RoboDK station: Config_2.rdk

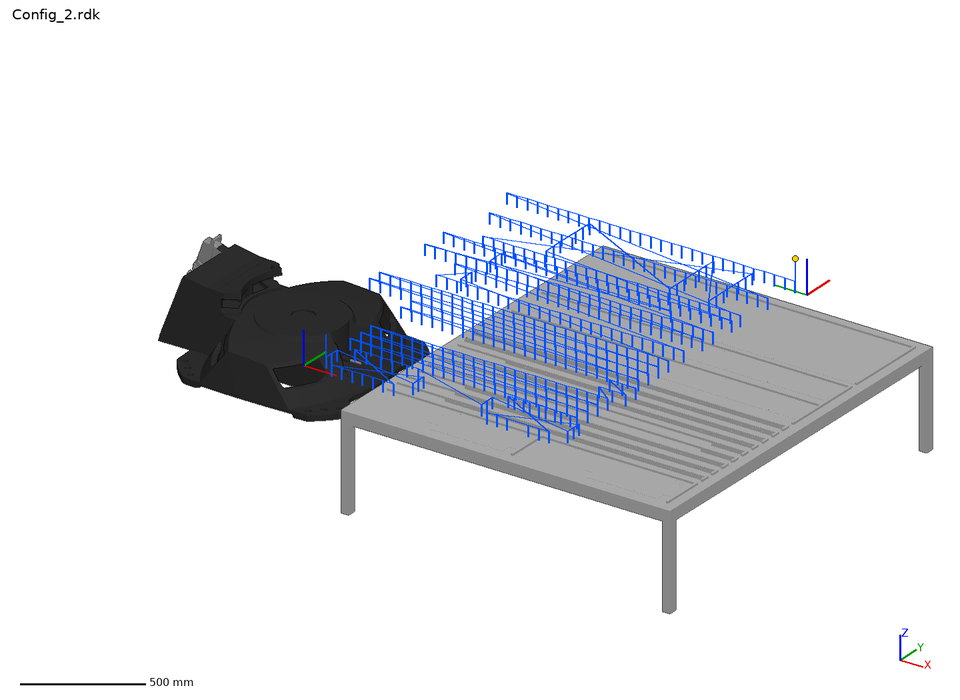
[picture v0: the station drawn from its stored meshes, robots at their saved joint values, targets as dots, program paths as lines]
Station Config_2 (saved by RoboDK 5.2.3). Poses are relative to the parent item; angles as X-Y-Z fixed-axis rotations.
  - frame KUKA KR 210 R2700 extra Base at (0, 0, 0) mm
    - robot KUKA KR 210 R2700 extra: 6 axes, payload 210 kg, reach 2696 mm, repeatability 0.06 mm, weight 1068 kg
        joint limits [-185, -140, -120, -350, -125, -350] to [185, -5, 155, 350, 125, 350]; home [0, -90, 90, 0, 0, 0]; saved at [44.26, -78.74, 122.767, 234.505, 59.006, -215.831]
      - tool Spindle, TCP at (278.6, 0, 88) mm, rotated rx 0 ry 90 rz 0 deg, size 85 x 346.5 x 128 mm
  - frame Corner First Plate at (1872.67, 817.07, 510.8) mm, rotated rx 0 ry 0 rz 90 deg
  - object Table 2 at (1700, -800, 455) mm, rotated rx 0 ry 0 rz 90 deg, size 1820 x 1600 x 475 mm, geometry from Table 2.stl
  - object Config_2 at (2495, 660, 510.8) mm, rotated rx 0 ry 0 rz 90 deg
  - machining project Path1 settings: rotZ(0) | rotX(0)*rotY(0) | rotz(0) | onStart | onPathStart | onApproach | onPoint | onRetract | onFinish | SetRPM(%1) | SetTool(%1) | Extruder(%1) | default | default | OutOnMov(%1) | OutOffMov(%1) | onPathFinish | M_RunCode(%1)
  - program Path1 (1338 instructions, listed below)
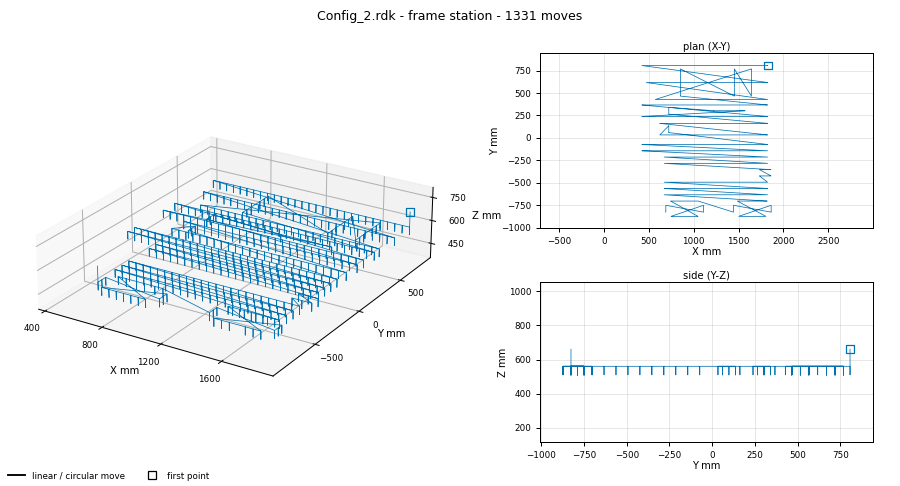
[picture p0: tool path of Config_2.rdk in frame station, 1331 of 1331 moves have a stored position in this frame; points joined in program order, loops and branches not executed]

--- program Path1 (robot KUKA KR 210 R2700 extra) ---
  Smooth(1)
  Set speed (1000.0 mm/s)
  Set Ref.: Corner First Plate
  Set Tool: Spindle
  Show Spindle
  MoveJ 1 to (-10.8, 50, 150) mm, rotated rx 180 ry 0 rz 90 deg; joints [-16.861, -44.669, 69.656, 144.341, 29.838, -148.103]
  MoveL 2 to (-10.8, 50, 150) mm, rotated rx 180 ry 0 rz 90 deg; joints [-16.861, -44.669, 69.656, 144.341, 29.838, -148.103]
  MoveL 3 to (-10.8, 50, 50) mm, rotated rx 180 ry 0 rz 90 deg; joints [-16.861, -42.157, 70.591, 147.522, 32.695, -151.823]
  MoveL 4 to (-10.8, 50, 50) mm, rotated rx 180 ry 0 rz 90 deg; joints [-16.861, -42.157, 70.591, 147.522, 32.695, -151.823]
  Set speed (150.0 mm/s)
  MoveL 5 to (-10.8, 50, -0.5) mm, rotated rx -180 ry 0 rz 90 deg; joints [-16.861, -40.791, 70.897, 148.859, 34.116, -153.424]
  MoveL 6 to (-10.8, 50, 50) mm, rotated rx 180 ry 0 rz 90 deg; joints [-16.861, -42.157, 70.591, 147.522, 32.695, -151.823]
  MoveL 7 to (-10.8, 100, 50) mm, rotated rx -180 ry 0 rz 90 deg; joints [-17.24, -44.27, 74.43, 148.298, 34.333, -152.976]
  MoveL 8 to (-10.8, 100, -0.5) mm, rotated rx -180 ry 0 rz 90 deg; joints [-17.24, -42.862, 74.73, 149.554, 35.795, -154.51]
  MoveL 9 to (-10.8, 100, 50) mm, rotated rx -180 ry 0 rz 90 deg; joints [-17.24, -44.27, 74.43, 148.298, 34.333, -152.976]
  MoveL 10 to (-10.8, 150, 50) mm, rotated rx -180 ry 0 rz 90 deg; joints [-17.637, -46.308, 78.104, 148.894, 35.906, -153.954]
  MoveL 11 to (-10.8, 150, -0.5) mm, rotated rx 180 ry 0 rz 90 deg; joints [-17.637, -44.857, 78.4, 150.085, 37.411, -155.439]
  MoveL 12 to (-10.8, 150, 50) mm, rotated rx -180 ry 0 rz 90 deg; joints [-17.637, -46.308, 78.104, 148.894, 35.906, -153.954]
  MoveL 13 to (-10.8, 200, 50) mm, rotated rx 180 ry 0 rz 90 deg; joints [-18.051, -48.282, 81.634, 149.341, 37.421, -154.79]
  MoveL 14 to (-10.8, 200, -0.5) mm, rotated rx -180 ry 0 rz 90 deg; joints [-18.051, -46.786, 81.927, 150.481, 38.968, -156.24]
  MoveL 15 to (-10.8, 200, 50) mm, rotated rx 180 ry 0 rz 90 deg; joints [-18.051, -48.282, 81.634, 149.341, 37.421, -154.79]
  MoveL 16 to (-10.8, 250, 50) mm, rotated rx 180 ry 0 rz 90 deg; joints [-18.485, -50.201, 85.037, 149.663, 38.882, -155.508]
  MoveL 17 to (-10.8, 250, -0.5) mm, rotated rx -180 ry 0 rz 90 deg; joints [-18.485, -48.66, 85.329, 150.761, 40.473, -156.934]
  MoveL 18 to (-10.8, 250, 50) mm, rotated rx 180 ry 0 rz 90 deg; joints [-18.485, -50.201, 85.037, 149.663, 38.882, -155.508]
  MoveL 19 to (-10.8, 300, 50) mm, rotated rx -180 ry 0 rz 90 deg; joints [-18.939, -52.073, 88.328, 149.877, 40.293, -156.128]
  MoveL 20 to (-10.8, 300, -0.5) mm, rotated rx 180 ry 0 rz 90 deg; joints [-18.939, -50.484, 88.62, 150.941, 41.929, -157.54]
  MoveL 21 to (-10.8, 300, 50) mm, rotated rx -180 ry 0 rz 90 deg; joints [-18.939, -52.073, 88.328, 149.877, 40.293, -156.128]
  MoveL 22 to (-10.8, 350, 50) mm, rotated rx 180 ry 0 rz 90 deg; joints [-19.415, -53.906, 91.518, 149.994, 41.659, -156.663]
  MoveL 23 to (-10.8, 350, -0.5) mm, rotated rx 180 ry 0 rz 90 deg; joints [-19.415, -52.267, 91.81, 151.032, 43.339, -158.069]
  MoveL 24 to (-10.8, 350, 50) mm, rotated rx 180 ry 0 rz 90 deg; joints [-19.415, -53.906, 91.518, 149.994, 41.659, -156.663]
  MoveL 25 to (-10.8, 400, 50) mm, rotated rx 180 ry 0 rz 90 deg; joints [-19.914, -55.704, 94.616, 150.026, 42.981, -157.123]
  MoveL 26 to (-10.8, 400, -0.5) mm, rotated rx -180 ry 0 rz 90 deg; joints [-19.914, -54.013, 94.91, 151.042, 44.709, -158.532]
  MoveL 27 to (-10.8, 400, 50) mm, rotated rx 180 ry 0 rz 90 deg; joints [-19.914, -55.704, 94.616, 150.026, 42.981, -157.123]
  MoveL 28 to (-10.8, 450, 50) mm, rotated rx 180 ry 0 rz 90 deg; joints [-20.439, -57.473, 97.631, 149.977, 44.262, -157.517]
  MoveL 29 to (-10.8, 450, -0.5) mm, rotated rx 180 ry 0 rz 90 deg; joints [-20.439, -55.727, 97.926, 150.978, 46.038, -158.936]
  MoveL 30 to (-10.8, 450, 50) mm, rotated rx 180 ry 0 rz 90 deg; joints [-20.439, -57.473, 97.631, 149.977, 44.262, -157.517]
  MoveL 31 to (-10.8, 500, 50) mm, rotated rx -180 ry 0 rz 90 deg; joints [-20.991, -59.217, 100.569, 149.854, 45.504, -157.852]
  MoveL 32 to (-10.8, 500, -0.5) mm, rotated rx 180 ry 0 rz 90 deg; joints [-20.991, -57.414, 100.867, 150.844, 47.331, -159.288]
  MoveL 33 to (-10.8, 500, 50) mm, rotated rx -180 ry 0 rz 90 deg; joints [-20.991, -59.217, 100.569, 149.854, 45.504, -157.852]
  MoveL 34 to (-10.8, 550, 50) mm, rotated rx 180 ry 0 rz 90 deg; joints [-21.572, -60.942, 103.435, 149.66, 46.709, -158.133]
  MoveL 35 to (-10.8, 550, -0.5) mm, rotated rx 180 ry 0 rz 90 deg; joints [-21.572, -59.078, 103.738, 150.643, 48.588, -159.592]
  MoveL 36 to (-10.8, 550, 50) mm, rotated rx 180 ry 0 rz 90 deg; joints [-21.572, -60.942, 103.435, 149.66, 46.709, -158.133]
  MoveL 37 to (-10.8, 600, 50) mm, rotated rx 180 ry 0 rz 90 deg; joints [-22.185, -62.649, 106.236, 149.397, 47.878, -158.362]
  MoveL 38 to (-10.8, 600, -0.5) mm, rotated rx 180 ry 0 rz 90 deg; joints [-22.185, -60.721, 106.543, 150.377, 49.812, -159.851]
  MoveL 39 to (-10.8, 600, 50) mm, rotated rx 180 ry 0 rz 90 deg; joints [-22.185, -62.649, 106.236, 149.397, 47.878, -158.362]
  MoveL 40 to (-10.8, 650, 50) mm, rotated rx 180 ry 0 rz 90 deg; joints [-22.832, -64.344, 108.975, 149.067, 49.013, -158.542]
  MoveL 41 to (-10.8, 650, -0.5) mm, rotated rx 180 ry 0 rz 90 deg; joints [-22.832, -62.348, 109.287, 150.048, 51.003, -160.069]
  MoveL 42 to (-10.8, 650, 50) mm, rotated rx 180 ry 0 rz 90 deg; joints [-22.832, -64.344, 108.975, 149.067, 49.013, -158.542]
  MoveL 43 to (-10.8, 700, 50) mm, rotated rx -180 ry 0 rz 90 deg; joints [-23.515, -66.029, 111.655, 148.669, 50.113, -158.676]
  MoveL 44 to (-10.8, 700, -0.5) mm, rotated rx 180 ry 0 rz 90 deg; joints [-23.515, -63.961, 111.973, 149.655, 52.163, -160.247]
  MoveL 45 to (-10.8, 700, 50) mm, rotated rx -180 ry 0 rz 90 deg; joints [-23.515, -66.029, 111.655, 148.669, 50.113, -158.676]
  MoveL 46 to (-10.8, 750, 50) mm, rotated rx 180 ry 0 rz 90 deg; joints [-24.238, -67.708, 114.279, 148.204, 51.181, -158.763]
  MoveL 47 to (-10.8, 750, -0.5) mm, rotated rx 180 ry 0 rz 90 deg; joints [-24.238, -65.564, 114.604, 149.198, 53.292, -160.386]
  MoveL 48 to (-10.8, 750, 50) mm, rotated rx 180 ry 0 rz 90 deg; joints [-24.238, -67.708, 114.279, 148.204, 51.181, -158.763]
  MoveL 49 to (-10.8, 800, 50) mm, rotated rx -180 ry 0 rz 90 deg; joints [-25.003, -69.384, 116.85, 147.669, 52.216, -158.805]
  MoveL 50 to (-10.8, 800, -0.5) mm, rotated rx 180 ry 0 rz 90 deg; joints [-25.003, -67.159, 117.183, 148.675, 54.391, -160.488]
  MoveL 51 to (-10.8, 800, 50) mm, rotated rx -180 ry 0 rz 90 deg; joints [-25.003, -69.384, 116.85, 147.669, 52.216, -158.805]
  MoveL 52 to (-10.8, 850, 50) mm, rotated rx -180 ry 0 rz 90 deg; joints [-25.816, -71.061, 119.369, 147.064, 53.22, -158.799]
  MoveL 53 to (-10.8, 850, -0.5) mm, rotated rx 180 ry 0 rz 90 deg; joints [-25.816, -68.749, 119.711, 148.085, 55.46, -160.551]
  MoveL 54 to (-10.8, 850, 50) mm, rotated rx -180 ry 0 rz 90 deg; joints [-25.816, -71.061, 119.369, 147.064, 53.22, -158.799]
  MoveL 55 to (-10.8, 900, 50) mm, rotated rx 180 ry 0 rz 90 deg; joints [-26.678, -72.742, 121.838, 146.383, 54.192, -158.746]
  MoveL 56 to (-10.8, 900, -0.5) mm, rotated rx -180 ry 0 rz 90 deg; joints [-26.678, -70.337, 122.19, 147.424, 56.501, -160.575]
  MoveL 57 to (-10.8, 900, 50) mm, rotated rx 180 ry 0 rz 90 deg; joints [-26.678, -72.742, 121.838, 146.383, 54.192, -158.746]
  MoveL 58 to (-10.8, 950, 50) mm, rotated rx -180 ry 0 rz 90 deg; joints [-27.596, -74.43, 124.259, 145.626, 55.132, -158.641]
  MoveL 59 to (-10.8, 950, -0.5) mm, rotated rx -180 ry 0 rz 90 deg; joints [-27.596, -71.926, 124.621, 146.689, 57.513, -160.559]
  MoveL 60 to (-10.8, 950, 50) mm, rotated rx -180 ry 0 rz 90 deg; joints [-27.596, -74.43, 124.259, 145.626, 55.132, -158.641]
  MoveL 61 to (-10.8, 1000, 50) mm, rotated rx 180 ry 0 rz 90 deg; joints [-28.574, -76.128, 126.631, 144.786, 56.043, -158.484]
  MoveL 62 to (-10.8, 1000, -0.5) mm, rotated rx 180 ry 0 rz 90 deg; joints [-28.574, -73.519, 127.005, 145.877, 58.497, -160.501]
  MoveL 63 to (-10.8, 1000, 50) mm, rotated rx 180 ry 0 rz 90 deg; joints [-28.574, -76.128, 126.631, 144.786, 56.043, -158.484]
  MoveL 64 to (-10.8, 1050, 50) mm, rotated rx -180 ry 0 rz 90 deg; joints [-29.617, -77.842, 128.955, 143.858, 56.923, -158.269]
  MoveL 65 to (-10.8, 1050, -0.5) mm, rotated rx 180 ry 0 rz 90 deg; joints [-29.617, -75.119, 129.342, 144.981, 59.453, -160.398]
  MoveL 66 to (-10.8, 1050, 50) mm, rotated rx -180 ry 0 rz 90 deg; joints [-29.617, -77.842, 128.955, 143.858, 56.923, -158.269]
  MoveL 67 to (-10.8, 1100, 50) mm, rotated rx 180 ry 0 rz 90 deg; joints [-30.732, -79.573, 131.231, 142.838, 57.775, -157.992]
  MoveL 68 to (-10.8, 1100, -0.5) mm, rotated rx -180 ry 0 rz 90 deg; joints [-30.732, -76.729, 131.632, 143.997, 60.382, -160.246]
  MoveL 69 to (-10.8, 1100, 50) mm, rotated rx 180 ry 0 rz 90 deg; joints [-30.732, -79.573, 131.231, 142.838, 57.775, -157.992]
  MoveL 70 to (-10.8, 1150, 50) mm, rotated rx 180 ry 0 rz 90 deg; joints [-31.924, -81.327, 133.457, 141.718, 58.599, -157.647]
  MoveL 71 to (-10.8, 1150, -0.5) mm, rotated rx 180 ry 0 rz 90 deg; joints [-31.924, -78.352, 133.874, 142.918, 61.284, -160.042]
  MoveL 72 to (-10.8, 1150, 50) mm, rotated rx 180 ry 0 rz 90 deg; joints [-31.924, -81.327, 133.457, 141.718, 58.599, -157.647]
  MoveL 73 to (-10.8, 1200, 50) mm, rotated rx 180 ry 0 rz 90 deg; joints [-33.202, -83.108, 135.634, 140.49, 59.397, -157.227]
  MoveL 74 to (-10.8, 1200, -0.5) mm, rotated rx 180 ry 0 rz 90 deg; joints [-33.202, -79.993, 136.068, 141.737, 62.161, -159.78]
  MoveL 75 to (-10.8, 1200, 50) mm, rotated rx 180 ry 0 rz 90 deg; joints [-33.202, -83.108, 135.634, 140.49, 59.397, -157.227]
  MoveL 76 to (-10.8, 1250, 50) mm, rotated rx -180 ry 0 rz 90 deg; joints [-34.574, -84.92, 137.758, 139.147, 60.172, -156.726]
  MoveL 77 to (-10.8, 1250, -0.5) mm, rotated rx -180 ry 0 rz 90 deg; joints [-34.574, -81.654, 138.211, 140.446, 63.014, -159.455]
  MoveL 78 to (-10.8, 1250, 50) mm, rotated rx -180 ry 0 rz 90 deg; joints [-34.574, -84.92, 137.758, 139.147, 60.172, -156.726]
  MoveL 79 to (-10.8, 1300, 50) mm, rotated rx 180 ry 0 rz 90 deg; joints [-36.047, -86.767, 139.828, 137.68, 60.929, -156.133]
  MoveL 80 to (-10.8, 1300, -0.5) mm, rotated rx 180 ry 0 rz 90 deg; joints [-36.047, -83.339, 140.302, 139.037, 63.846, -159.059]
  MoveL 81 to (-10.8, 1300, 50) mm, rotated rx 180 ry 0 rz 90 deg; joints [-36.047, -86.767, 139.828, 137.68, 60.929, -156.133]
  MoveL 82 to (-10.8, 1350, 50) mm, rotated rx 180 ry 0 rz 90 deg; joints [-37.633, -88.655, 141.842, 136.078, 61.671, -155.439]
  MoveL 83 to (-10.8, 1350, -0.5) mm, rotated rx 180 ry 0 rz 90 deg; joints [-37.633, -85.052, 142.339, 137.499, 64.659, -158.585]
  MoveL 84 to (-10.8, 1350, 50) mm, rotated rx 180 ry 0 rz 90 deg; joints [-37.633, -88.655, 141.842, 136.078, 61.671, -155.439]
  MoveL 85 to (-10.8, 1400, 50) mm, rotated rx -180 ry 0 rz 90 deg; joints [-39.341, -90.587, 143.795, 134.333, 62.407, -154.634]
  MoveL 86 to (-10.8, 1400, -0.5) mm, rotated rx 180 ry 0 rz 90 deg; joints [-39.341, -86.798, 144.317, 135.822, 65.461, -158.023]
  MoveL 87 to (-10.8, 1400, 50) mm, rotated rx -180 ry 0 rz 90 deg; joints [-39.341, -90.587, 143.795, 134.333, 62.407, -154.634]
  MoveL 88 to (-10.8, 1450, 50) mm, rotated rx 180 ry 0 rz 90 deg; joints [-41.184, -92.567, 145.684, 132.434, 63.147, -153.707]
  MoveL 89 to (-10.8, 1450, -0.5) mm, rotated rx -180 ry 0 rz 90 deg; joints [-41.184, -88.578, 146.233, 133.998, 66.256, -157.364]
  MoveL 90 to (-10.8, 1450, 50) mm, rotated rx 180 ry 0 rz 90 deg; joints [-41.184, -92.567, 145.684, 132.434, 63.147, -153.707]
  MoveL 91 to (-200, 50, 50) mm, rotated rx -180 ry 0 rz 90 deg; joints [-12.12, -44.252, 74.397, 156.847, 32.277, -160.122]
  MoveL 92 to (-200, 50, -0.5) mm, rotated rx -180 ry 0 rz 90 deg; joints [-12.12, -42.844, 74.697, 157.857, 33.853, -161.328]
  MoveL 93 to (-200, 50, 50) mm, rotated rx -180 ry 0 rz 90 deg; joints [-12.12, -44.252, 74.397, 156.847, 32.277, -160.122]
  MoveL 94 to (-200, 100, 50) mm, rotated rx 180 ry 0 rz 90 deg; joints [-12.401, -46.339, 78.159, 157.362, 33.914, -160.91]
  MoveL 95 to (-200, 100, -0.5) mm, rotated rx 180 ry 0 rz 90 deg; joints [-12.401, -44.887, 78.455, 158.313, 35.532, -162.067]
  MoveL 96 to (-200, 100, 50) mm, rotated rx 180 ry 0 rz 90 deg; joints [-12.401, -46.339, 78.159, 157.362, 33.914, -160.91]
  MoveL 97 to (-200, 150, 50) mm, rotated rx 180 ry 0 rz 90 deg; joints [-12.695, -48.361, 81.776, 157.752, 35.481, -161.577]
  MoveL 98 to (-200, 150, -0.5) mm, rotated rx -180 ry 0 rz 90 deg; joints [-12.695, -46.864, 82.069, 158.657, 37.144, -162.699]
  MoveL 99 to (-200, 150, 50) mm, rotated rx 180 ry 0 rz 90 deg; joints [-12.695, -48.361, 81.776, 157.752, 35.481, -161.577]
  MoveL 100 to (-200, 200, 50) mm, rotated rx -180 ry 0 rz 90 deg; joints [-13.003, -50.329, 85.264, 158.038, 36.986, -162.145]
  MoveL 101 to (-200, 200, -0.5) mm, rotated rx -180 ry 0 rz 90 deg; joints [-13.003, -48.785, 85.556, 158.905, 38.694, -163.244]
  MoveL 102 to (-200, 200, 50) mm, rotated rx -180 ry 0 rz 90 deg; joints [-13.003, -50.329, 85.264, 158.038, 36.986, -162.145]
  MoveL 103 to (-200, 250, 50) mm, rotated rx -180 ry 0 rz 90 deg; joints [-13.326, -52.251, 88.639, 158.234, 38.432, -162.632]
  MoveL 104 to (-200, 250, -0.5) mm, rotated rx 180 ry 0 rz 90 deg; joints [-13.326, -50.658, 88.93, 159.072, 40.188, -163.715]
  MoveL 105 to (-200, 250, 50) mm, rotated rx -180 ry 0 rz 90 deg; joints [-13.326, -52.251, 88.639, 158.234, 38.432, -162.632]
  MoveL 106 to (-200, 300, 50) mm, rotated rx 180 ry 0 rz 90 deg; joints [-13.665, -54.134, 91.913, 158.353, 39.825, -163.049]
  MoveL 107 to (-200, 300, -0.5) mm, rotated rx 180 ry 0 rz 90 deg; joints [-13.665, -52.489, 92.205, 159.169, 41.63, -164.124]
  MoveL 108 to (-200, 300, 50) mm, rotated rx 180 ry 0 rz 90 deg; joints [-13.665, -54.134, 91.913, 158.353, 39.825, -163.049]
  MoveL 109 to (-200, 350, 50) mm, rotated rx 180 ry 0 rz 90 deg; joints [-14.022, -55.984, 95.096, 158.403, 41.167, -163.405]
  MoveL 110 to (-200, 350, -0.5) mm, rotated rx -180 ry 0 rz 90 deg; joints [-14.022, -54.285, 95.39, 159.201, 43.025, -164.48]
  MoveL 111 to (-200, 350, 50) mm, rotated rx 180 ry 0 rz 90 deg; joints [-14.022, -55.984, 95.096, 158.403, 41.167, -163.405]
  MoveL 112 to (-200, 400, 50) mm, rotated rx -180 ry 0 rz 90 deg; joints [-14.397, -57.808, 98.197, 158.389, 42.461, -163.709]
  MoveL 113 to (-200, 400, -0.5) mm, rotated rx 180 ry 0 rz 90 deg; joints [-14.397, -56.051, 98.494, 159.174, 44.374, -164.79]
  MoveL 114 to (-200, 400, 50) mm, rotated rx -180 ry 0 rz 90 deg; joints [-14.397, -57.808, 98.197, 158.389, 42.461, -163.709]
  MoveL 115 to (-200, 450, 50) mm, rotated rx 180 ry 0 rz 90 deg; joints [-14.792, -59.609, 101.223, 158.316, 43.709, -163.964]
  MoveL 116 to (-200, 450, -0.5) mm, rotated rx 180 ry 0 rz 90 deg; joints [-14.792, -57.793, 101.523, 159.093, 45.681, -165.057]
  MoveL 117 to (-200, 450, 50) mm, rotated rx 180 ry 0 rz 90 deg; joints [-14.792, -59.609, 101.223, 158.316, 43.709, -163.964]
  MoveL 118 to (-200, 500, 50) mm, rotated rx 180 ry 0 rz 90 deg; joints [-15.209, -61.394, 104.181, 158.187, 44.913, -164.175]
  MoveL 119 to (-200, 500, -0.5) mm, rotated rx 180 ry 0 rz 90 deg; joints [-15.209, -59.513, 104.485, 158.96, 46.946, -165.286]
  MoveL 120 to (-200, 500, 50) mm, rotated rx 180 ry 0 rz 90 deg; joints [-15.209, -61.394, 104.181, 158.187, 44.913, -164.175]
  MoveL 121 to (-200, 550, 50) mm, rotated rx 180 ry 0 rz 90 deg; joints [-15.65, -63.166, 107.075, 158.004, 46.074, -164.346]
  MoveL 122 to (-200, 550, -0.5) mm, rotated rx 180 ry 0 rz 90 deg; joints [-15.65, -61.217, 107.384, 158.776, 48.172, -165.48]
  MoveL 123 to (-200, 550, 50) mm, rotated rx 180 ry 0 rz 90 deg; joints [-15.65, -63.166, 107.075, 158.004, 46.074, -164.346]
  MoveL 124 to (-200, 600, 50) mm, rotated rx 180 ry 0 rz 90 deg; joints [-16.116, -64.929, 109.91, 157.767, 47.192, -164.476]
  MoveL 125 to (-200, 600, -0.5) mm, rotated rx -180 ry 0 rz 90 deg; joints [-16.116, -62.909, 110.225, 158.542, 49.36, -165.64]
  MoveL 126 to (-200, 600, 50) mm, rotated rx 180 ry 0 rz 90 deg; joints [-16.116, -64.929, 109.91, 157.767, 47.192, -164.476]
  MoveL 127 to (-200, 650, 50) mm, rotated rx -180 ry 0 rz 90 deg; joints [-16.611, -66.688, 112.691, 157.477, 48.268, -164.569]
  MoveL 128 to (-200, 650, -0.5) mm, rotated rx -180 ry 0 rz 90 deg; joints [-16.611, -64.591, 113.012, 158.258, 50.509, -165.769]
  MoveL 129 to (-200, 650, 50) mm, rotated rx -180 ry 0 rz 90 deg; joints [-16.611, -66.688, 112.691, 157.477, 48.268, -164.569]
  MoveL 130 to (-200, 700, 50) mm, rotated rx 180 ry 0 rz 90 deg; joints [-17.135, -68.448, 115.42, 157.132, 49.302, -164.623]
  MoveL 131 to (-200, 700, -0.5) mm, rotated rx 180 ry 0 rz 90 deg; joints [-17.135, -66.269, 115.749, 157.924, 51.62, -165.866]
  MoveL 132 to (-200, 700, 50) mm, rotated rx 180 ry 0 rz 90 deg; joints [-17.135, -68.448, 115.42, 157.132, 49.302, -164.623]
  MoveL 133 to (-200, 750, 50) mm, rotated rx 180 ry 0 rz 90 deg; joints [-17.693, -70.213, 118.101, 156.732, 50.293, -164.639]
  MoveL 134 to (-200, 750, -0.5) mm, rotated rx -180 ry 0 rz 90 deg; joints [-17.693, -67.945, 118.438, 157.537, 52.694, -165.932]
  MoveL 135 to (-200, 750, 50) mm, rotated rx 180 ry 0 rz 90 deg; joints [-17.693, -70.213, 118.101, 156.732, 50.293, -164.639]
  MoveL 136 to (-200, 800, 50) mm, rotated rx 180 ry 0 rz 90 deg; joints [-18.287, -71.986, 120.735, 156.273, 51.24, -164.614]
  MoveL 137 to (-200, 800, -0.5) mm, rotated rx -180 ry 0 rz 90 deg; joints [-18.287, -69.624, 121.082, 157.096, 53.729, -165.966]
  MoveL 138 to (-200, 800, 50) mm, rotated rx 180 ry 0 rz 90 deg; joints [-18.287, -71.986, 120.735, 156.273, 51.24, -164.614]
  MoveL 139 to (-200, 850, 50) mm, rotated rx 180 ry 0 rz 90 deg; joints [-18.92, -73.774, 123.326, 155.752, 52.142, -164.548]
  MoveL 140 to (-200, 850, -0.5) mm, rotated rx 180 ry 0 rz 90 deg; joints [-18.92, -71.309, 123.684, 156.598, 54.724, -165.967]
  MoveL 141 to (-200, 850, 50) mm, rotated rx 180 ry 0 rz 90 deg; joints [-18.92, -73.774, 123.326, 155.752, 52.142, -164.548]
  MoveL 142 to (-200, 900, 50) mm, rotated rx 180 ry 0 rz 90 deg; joints [-19.598, -75.582, 125.874, 155.166, 52.997, -164.436]
  MoveL 143 to (-200, 900, -0.5) mm, rotated rx -180 ry 0 rz 90 deg; joints [-19.598, -73.007, 126.245, 156.039, 55.679, -165.933]
  MoveL 144 to (-200, 900, 50) mm, rotated rx 180 ry 0 rz 90 deg; joints [-19.598, -75.582, 125.874, 155.166, 52.997, -164.436]
  MoveL 145 to (-200, 950, 50) mm, rotated rx -180 ry 0 rz 90 deg; joints [-20.323, -77.414, 128.382, 154.508, 53.803, -164.274]
  MoveL 146 to (-200, 950, -0.5) mm, rotated rx 180 ry 0 rz 90 deg; joints [-20.323, -74.72, 128.765, 155.414, 56.592, -165.86]
  MoveL 147 to (-200, 950, 50) mm, rotated rx -180 ry 0 rz 90 deg; joints [-20.323, -77.414, 128.382, 154.508, 53.803, -164.274]
  MoveL 148 to (-200, 1000, 50) mm, rotated rx 180 ry 0 rz 90 deg; joints [-21.102, -79.279, 130.849, 153.774, 54.558, -164.057]
  MoveL 149 to (-200, 1000, -0.5) mm, rotated rx 180 ry 0 rz 90 deg; joints [-21.102, -76.456, 131.248, 154.718, 57.46, -165.746]
  MoveL 150 to (-200, 1000, 50) mm, rotated rx 180 ry 0 rz 90 deg; joints [-21.102, -79.279, 130.849, 153.774, 54.558, -164.057]
  MoveL 151 to (-200, 1050, 50) mm, rotated rx -180 ry 0 rz 90 deg; joints [-21.94, -81.183, 133.277, 152.955, 55.258, -163.779]
  MoveL 152 to (-200, 1050, -0.5) mm, rotated rx 180 ry 0 rz 90 deg; joints [-21.94, -78.219, 133.692, 153.945, 58.282, -165.585]
  MoveL 153 to (-200, 1050, 50) mm, rotated rx -180 ry 0 rz 90 deg; joints [-21.94, -81.183, 133.277, 152.955, 55.258, -163.779]
  MoveL 154 to (-200, 1100, 50) mm, rotated rx 180 ry 0 rz 90 deg; joints [-22.843, -83.135, 135.665, 152.043, 55.901, -163.429]
  MoveL 155 to (-200, 1100, -0.5) mm, rotated rx 180 ry 0 rz 90 deg; joints [-22.843, -80.017, 136.1, 153.087, 59.054, -165.37]
  MoveL 156 to (-200, 1100, 50) mm, rotated rx 180 ry 0 rz 90 deg; joints [-22.843, -83.135, 135.665, 152.043, 55.901, -163.429]
  MoveL 157 to (-200, 1150, 50) mm, rotated rx 180 ry 0 rz 90 deg; joints [-23.819, -85.144, 138.014, 151.026, 56.481, -162.998]
  MoveL 158 to (-200, 1150, -0.5) mm, rotated rx -180 ry 0 rz 90 deg; joints [-23.819, -81.858, 138.469, 152.134, 59.772, -165.095]
  MoveL 159 to (-200, 1150, 50) mm, rotated rx 180 ry 0 rz 90 deg; joints [-23.819, -85.144, 138.014, 151.026, 56.481, -162.998]
  MoveL 160 to (-200, 1200, 50) mm, rotated rx 180 ry 0 rz 90 deg; joints [-24.878, -87.221, 140.322, 149.892, 56.996, -162.471]
  MoveL 161 to (-200, 1200, -0.5) mm, rotated rx 180 ry 0 rz 90 deg; joints [-24.878, -83.751, 140.801, 151.075, 60.433, -164.747]
  MoveL 162 to (-200, 1200, 50) mm, rotated rx 180 ry 0 rz 90 deg; joints [-24.878, -87.221, 140.322, 149.892, 56.996, -162.471]
  MoveL 163 to (-200, 1250, 50) mm, rotated rx 180 ry 0 rz 90 deg; joints [-26.027, -89.38, 142.587, 148.626, 57.441, -161.832]
  MoveL 164 to (-200, 1250, -0.5) mm, rotated rx 180 ry 0 rz 90 deg; joints [-26.027, -85.708, 143.093, 149.897, 61.032, -164.316]
  MoveL 165 to (-200, 1250, 50) mm, rotated rx 180 ry 0 rz 90 deg; joints [-26.027, -89.38, 142.587, 148.626, 57.441, -161.832]
  MoveL 166 to (-200, 1300, 50) mm, rotated rx -180 ry 0 rz 90 deg; joints [-27.28, -91.635, 144.809, 147.209, 57.811, -161.058]
  MoveL 167 to (-200, 1300, -0.5) mm, rotated rx -180 ry 0 rz 90 deg; joints [-27.28, -87.741, 145.345, 148.586, 61.564, -163.784]
  MoveL 168 to (-200, 1300, 50) mm, rotated rx -180 ry 0 rz 90 deg; joints [-27.28, -91.635, 144.809, 147.209, 57.811, -161.058]
  MoveL 169 to (-200, 1350, 50) mm, rotated rx -180 ry 0 rz 90 deg; joints [-28.649, -94.005, 146.985, 145.618, 58.103, -160.123]
  MoveL 170 to (-200, 1350, -0.5) mm, rotated rx 180 ry 0 rz 90 deg; joints [-28.649, -89.867, 147.555, 147.121, 62.025, -163.131]
  MoveL 171 to (-200, 1350, 50) mm, rotated rx -180 ry 0 rz 90 deg; joints [-28.649, -94.005, 146.985, 145.618, 58.103, -160.123]
  MoveL 172 to (-200, 1400, 50) mm, rotated rx -180 ry 0 rz 90 deg; joints [-30.148, -96.511, 149.11, 143.828, 58.316, -158.993]
  MoveL 173 to (-200, 1400, -0.5) mm, rotated rx -180 ry 0 rz 90 deg; joints [-30.148, -92.103, 149.718, 145.481, 62.41, -162.331]
  MoveL 174 to (-200, 1400, 50) mm, rotated rx -180 ry 0 rz 90 deg; joints [-30.148, -96.511, 149.11, 143.828, 58.316, -158.993]
  MoveL 175 to (-389.2, 50, 50) mm, rotated rx 180 ry 0 rz 90 deg; joints [-7.205, -45.617, 76.862, 166.302, 31.983, -168.319]
  MoveL 176 to (-389.2, 50, -0.5) mm, rotated rx -180 ry 0 rz 90 deg; joints [-7.205, -44.181, 77.159, 166.924, 33.669, -169.06]
  MoveL 177 to (-389.2, 50, 50) mm, rotated rx 180 ry 0 rz 90 deg; joints [-7.205, -45.617, 76.862, 166.302, 31.983, -168.319]
  MoveL 178 to (-389.2, 100, 50) mm, rotated rx 180 ry 0 rz 90 deg; joints [-7.376, -47.693, 80.584, 166.593, 33.617, -168.772]
  MoveL 179 to (-389.2, 100, -0.5) mm, rotated rx 180 ry 0 rz 90 deg; joints [-7.376, -46.211, 80.878, 167.179, 35.346, -169.484]
  MoveL 180 to (-389.2, 100, 50) mm, rotated rx 180 ry 0 rz 90 deg; joints [-7.376, -47.693, 80.584, 166.593, 33.617, -168.772]
  MoveL 181 to (-389.2, 150, 50) mm, rotated rx 180 ry 0 rz 90 deg; joints [-7.554, -49.71, 84.17, 166.81, 35.178, -169.155]
  MoveL 182 to (-389.2, 150, -0.5) mm, rotated rx -180 ry 0 rz 90 deg; joints [-7.554, -48.181, 84.462, 167.368, 36.953, -169.847]
  MoveL 183 to (-389.2, 150, 50) mm, rotated rx 180 ry 0 rz 90 deg; joints [-7.554, -49.71, 84.17, 166.81, 35.178, -169.155]
  MoveL 184 to (-389.2, 200, 50) mm, rotated rx -180 ry 0 rz 90 deg; joints [-7.742, -51.679, 87.638, 166.965, 36.673, -169.481]
  MoveL 185 to (-389.2, 200, -0.5) mm, rotated rx 180 ry 0 rz 90 deg; joints [-7.742, -50.101, 87.93, 167.502, 38.496, -170.158]
  MoveL 186 to (-389.2, 200, 50) mm, rotated rx -180 ry 0 rz 90 deg; joints [-7.742, -51.679, 87.638, 166.965, 36.673, -169.481]
  MoveL 187 to (-389.2, 250, 50) mm, rotated rx -180 ry 0 rz 90 deg; joints [-7.938, -53.608, 91.001, 167.068, 38.106, -169.758]
  MoveL 188 to (-389.2, 250, -0.5) mm, rotated rx 180 ry 0 rz 90 deg; joints [-7.938, -51.977, 91.293, 167.588, 39.982, -170.428]
  MoveL 189 to (-389.2, 250, 50) mm, rotated rx -180 ry 0 rz 90 deg; joints [-7.938, -53.608, 91.001, 167.068, 38.106, -169.758]
  MoveL 190 to (-389.2, 300, 50) mm, rotated rx -180 ry 0 rz 90 deg; joints [-8.145, -55.502, 94.27, 167.125, 39.482, -169.995]
  MoveL 191 to (-389.2, 300, -0.5) mm, rotated rx -180 ry 0 rz 90 deg; joints [-8.145, -53.818, 94.564, 167.632, 41.413, -170.661]
  MoveL 192 to (-389.2, 300, 50) mm, rotated rx -180 ry 0 rz 90 deg; joints [-8.145, -55.502, 94.27, 167.125, 39.482, -169.995]
  MoveL 193 to (-389.2, 350, 50) mm, rotated rx 180 ry 0 rz 90 deg; joints [-8.363, -57.369, 97.455, 167.139, 40.804, -170.195]
  MoveL 194 to (-389.2, 350, -0.5) mm, rotated rx 180 ry 0 rz 90 deg; joints [-8.363, -55.627, 97.751, 167.637, 42.793, -170.863]
  MoveL 195 to (-389.2, 350, 50) mm, rotated rx 180 ry 0 rz 90 deg; joints [-8.363, -57.369, 97.455, 167.139, 40.804, -170.195]
  MoveL 196 to (-389.2, 400, 50) mm, rotated rx 180 ry 0 rz 90 deg; joints [-8.593, -59.215, 100.564, 167.116, 42.075, -170.364]
  MoveL 197 to (-389.2, 400, -0.5) mm, rotated rx 180 ry 0 rz 90 deg; joints [-8.593, -57.412, 100.863, 167.607, 44.126, -171.037]
  MoveL 198 to (-389.2, 400, 50) mm, rotated rx 180 ry 0 rz 90 deg; joints [-8.593, -59.215, 100.564, 167.116, 42.075, -170.364]
  MoveL 199 to (-389.2, 450, 50) mm, rotated rx -180 ry 0 rz 90 deg; joints [-8.836, -61.043, 103.603, 167.056, 43.295, -170.503]
  MoveL 200 to (-389.2, 450, -0.5) mm, rotated rx -180 ry 0 rz 90 deg; joints [-8.836, -59.176, 103.906, 167.544, 45.413, -171.186]
  MoveL 201 to (-389.2, 450, 50) mm, rotated rx -180 ry 0 rz 90 deg; joints [-8.836, -61.043, 103.603, 167.056, 43.295, -170.503]
  MoveL 202 to (-389.2, 500, 50) mm, rotated rx 180 ry 0 rz 90 deg; joints [-9.093, -62.86, 106.579, 166.962, 44.467, -170.616]
  MoveL 203 to (-389.2, 500, -0.5) mm, rotated rx -180 ry 0 rz 90 deg; joints [-9.093, -60.924, 106.887, 167.449, 46.655, -171.312]
  MoveL 204 to (-389.2, 500, 50) mm, rotated rx 180 ry 0 rz 90 deg; joints [-9.093, -62.86, 106.579, 166.962, 44.467, -170.616]
  MoveL 205 to (-389.2, 550, 50) mm, rotated rx -180 ry 0 rz 90 deg; joints [-9.365, -64.67, 109.497, 166.833, 45.59, -170.703]
  MoveL 206 to (-389.2, 550, -0.5) mm, rotated rx 180 ry 0 rz 90 deg; joints [-9.365, -62.661, 109.811, 167.322, 47.855, -171.416]
  MoveL 207 to (-389.2, 550, 50) mm, rotated rx -180 ry 0 rz 90 deg; joints [-9.365, -64.67, 109.497, 166.833, 45.59, -170.703]
  MoveL 208 to (-389.2, 600, 50) mm, rotated rx -180 ry 0 rz 90 deg; joints [-9.654, -66.479, 112.362, 166.67, 46.665, -170.765]
  MoveL 209 to (-389.2, 600, -0.5) mm, rotated rx -180 ry 0 rz 90 deg; joints [-9.654, -64.391, 112.682, 167.164, 49.011, -171.5]
  MoveL 210 to (-389.2, 600, 50) mm, rotated rx -180 ry 0 rz 90 deg; joints [-9.654, -66.479, 112.362, 166.67, 46.665, -170.765]
  MoveL 211 to (-389.2, 650, 50) mm, rotated rx -180 ry 0 rz 90 deg; joints [-9.96, -68.29, 115.177, 166.473, 47.69, -170.802]
  MoveL 212 to (-389.2, 650, -0.5) mm, rotated rx -180 ry 0 rz 90 deg; joints [-9.96, -66.118, 115.505, 166.974, 50.123, -171.563]
  MoveL 213 to (-389.2, 650, 50) mm, rotated rx -180 ry 0 rz 90 deg; joints [-9.96, -68.29, 115.177, 166.473, 47.69, -170.802]
  MoveL 214 to (-389.2, 700, 50) mm, rotated rx 180 ry 0 rz 90 deg; joints [-10.287, -70.109, 117.945, 166.241, 48.665, -170.813]
  MoveL 215 to (-389.2, 700, -0.5) mm, rotated rx 180 ry 0 rz 90 deg; joints [-10.287, -67.847, 118.282, 166.752, 51.192, -171.607]
  MoveL 216 to (-389.2, 700, 50) mm, rotated rx 180 ry 0 rz 90 deg; joints [-10.287, -70.109, 117.945, 166.241, 48.665, -170.813]
  MoveL 217 to (-389.2, 750, 50) mm, rotated rx 180 ry 0 rz 90 deg; joints [-10.636, -71.942, 120.671, 165.971, 49.587, -170.799]
  MoveL 218 to (-389.2, 750, -0.5) mm, rotated rx -180 ry 0 rz 90 deg; joints [-10.636, -69.582, 121.018, 166.495, 52.216, -171.629]
  MoveL 219 to (-389.2, 750, 50) mm, rotated rx 180 ry 0 rz 90 deg; joints [-10.636, -71.942, 120.671, 165.971, 49.587, -170.799]
  MoveL 220 to (-389.2, 800, 50) mm, rotated rx 180 ry 0 rz 90 deg; joints [-11.009, -73.795, 123.356, 165.662, 50.454, -170.756]
  MoveL 221 to (-389.2, 800, -0.5) mm, rotated rx 180 ry 0 rz 90 deg; joints [-11.009, -71.329, 123.714, 166.202, 53.193, -171.63]
  MoveL 222 to (-389.2, 800, 50) mm, rotated rx 180 ry 0 rz 90 deg; joints [-11.009, -73.795, 123.356, 165.662, 50.454, -170.756]
  MoveL 223 to (-389.2, 850, 50) mm, rotated rx -180 ry 0 rz 90 deg; joints [-11.408, -75.674, 126.003, 165.31, 51.262, -170.684]
  MoveL 224 to (-389.2, 850, -0.5) mm, rotated rx 180 ry 0 rz 90 deg; joints [-11.408, -73.093, 126.374, 165.87, 54.12, -171.607]
  MoveL 225 to (-389.2, 850, 50) mm, rotated rx -180 ry 0 rz 90 deg; joints [-11.408, -75.674, 126.003, 165.31, 51.262, -170.684]
  MoveL 226 to (-389.2, 900, 50) mm, rotated rx 180 ry 0 rz 90 deg; joints [-11.838, -77.587, 128.614, 164.912, 52.006, -170.577]
  MoveL 227 to (-389.2, 900, -0.5) mm, rotated rx -180 ry 0 rz 90 deg; joints [-11.838, -74.881, 128.999, 165.496, 54.994, -171.559]
  MoveL 228 to (-389.2, 900, 50) mm, rotated rx 180 ry 0 rz 90 deg; joints [-11.838, -77.587, 128.614, 164.912, 52.006, -170.577]
  MoveL 229 to (-389.2, 950, 50) mm, rotated rx 180 ry 0 rz 90 deg; joints [-12.3, -79.542, 131.19, 164.462, 52.681, -170.432]
  MoveL 230 to (-389.2, 950, -0.5) mm, rotated rx 180 ry 0 rz 90 deg; joints [-12.3, -76.7, 131.591, 165.076, 55.811, -171.482]
  MoveL 231 to (-389.2, 950, 50) mm, rotated rx 180 ry 0 rz 90 deg; joints [-12.3, -79.542, 131.19, 164.462, 52.681, -170.432]
  MoveL 232 to (-389.2, 1000, 50) mm, rotated rx -180 ry 0 rz 90 deg; joints [-12.799, -81.549, 133.733, 163.956, 53.28, -170.244]
  MoveL 233 to (-389.2, 1000, -0.5) mm, rotated rx 180 ry 0 rz 90 deg; joints [-12.799, -78.557, 134.152, 164.605, 56.564, -171.373]
  MoveL 234 to (-389.2, 1000, 50) mm, rotated rx -180 ry 0 rz 90 deg; joints [-12.799, -81.549, 133.733, 163.956, 53.28, -170.244]
  MoveL 235 to (-389.2, 1050, 50) mm, rotated rx 180 ry 0 rz 90 deg; joints [-13.34, -83.621, 136.243, 163.385, 53.795, -170.004]
  MoveL 236 to (-389.2, 1050, -0.5) mm, rotated rx -180 ry 0 rz 90 deg; joints [-13.34, -80.463, 136.683, 164.077, 57.248, -171.226]
  MoveL 237 to (-389.2, 1050, 50) mm, rotated rx 180 ry 0 rz 90 deg; joints [-13.34, -83.621, 136.243, 163.385, 53.795, -170.004]
  MoveL 238 to (-389.2, 1100, 50) mm, rotated rx -180 ry 0 rz 90 deg; joints [-13.928, -85.77, 138.722, 162.74, 54.214, -169.702]
  MoveL 239 to (-389.2, 1100, -0.5) mm, rotated rx -180 ry 0 rz 90 deg; joints [-13.928, -82.43, 139.185, 163.484, 57.852, -171.034]
  MoveL 240 to (-389.2, 1100, 50) mm, rotated rx -180 ry 0 rz 90 deg; joints [-13.928, -85.77, 138.722, 162.74, 54.214, -169.702]
  MoveL 241 to (-389.2, 1150, 50) mm, rotated rx 180 ry 0 rz 90 deg; joints [-14.568, -88.014, 141.17, 162.009, 54.524, -169.327]
  MoveL 242 to (-389.2, 1150, -0.5) mm, rotated rx 180 ry 0 rz 90 deg; joints [-14.568, -84.471, 141.658, 162.817, 58.367, -170.788]
  MoveL 243 to (-389.2, 1150, 50) mm, rotated rx 180 ry 0 rz 90 deg; joints [-14.568, -88.014, 141.17, 162.009, 54.524, -169.327]
  MoveL 244 to (-389.2, 1200, 50) mm, rotated rx -180 ry 0 rz 90 deg; joints [-15.269, -90.374, 143.585, 161.177, 54.709, -168.859]
  MoveL 245 to (-389.2, 1200, -0.5) mm, rotated rx -180 ry 0 rz 90 deg; joints [-15.269, -86.606, 144.104, 162.064, 58.778, -170.476]
  MoveL 246 to (-389.2, 1200, 50) mm, rotated rx -180 ry 0 rz 90 deg; joints [-15.269, -90.374, 143.585, 161.177, 54.709, -168.859]
  MoveL 247 to (-389.2, 1250, 50) mm, rotated rx 180 ry 0 rz 90 deg; joints [-16.039, -92.875, 145.968, 160.226, 54.75, -168.278]
  MoveL 248 to (-389.2, 1250, -0.5) mm, rotated rx 180 ry 0 rz 90 deg; joints [-16.039, -88.855, 146.522, 161.21, 59.068, -170.08]
  MoveL 249 to (-389.2, 1250, 50) mm, rotated rx 180 ry 0 rz 90 deg; joints [-16.039, -92.875, 145.968, 160.226, 54.75, -168.278]
  MoveL 250 to (-389.2, 1300, 50) mm, rotated rx -180 ry 0 rz 90 deg; joints [-16.888, -95.552, 148.317, 159.128, 54.621, -167.55]
  MoveL 251 to (-389.2, 1300, -0.5) mm, rotated rx -180 ry 0 rz 90 deg; joints [-16.888, -91.248, 148.91, 160.236, 59.214, -169.579]
  MoveL 252 to (-389.2, 1300, 50) mm, rotated rx -180 ry 0 rz 90 deg; joints [-16.888, -95.552, 148.317, 159.128, 54.621, -167.55]
  MoveL 253 to (-48.6, 230, 50) mm, rotated rx -180 ry 0 rz 90 deg; joints [-17.308, -49.904, 84.513, 151.248, 38.207, -156.678]
  MoveL 254 to (-48.6, 230, -0.5) mm, rotated rx 180 ry 0 rz 90 deg; joints [-17.308, -48.37, 84.805, 152.314, 39.816, -158.049]
  MoveL 255 to (-48.6, 230, 50) mm, rotated rx -180 ry 0 rz 90 deg; joints [-17.308, -49.904, 84.513, 151.248, 38.207, -156.678]
  MoveL 256 to (-98.6, 230, 50) mm, rotated rx -180 ry 0 rz 90 deg; joints [-15.968, -50.476, 85.523, 153.514, 38.085, -158.585]
  MoveL 257 to (-98.6, 230, -0.5) mm, rotated rx 180 ry 0 rz 90 deg; joints [-15.968, -48.928, 85.815, 154.512, 39.739, -159.868]
  MoveL 258 to (-98.6, 230, 50) mm, rotated rx -180 ry 0 rz 90 deg; joints [-15.968, -50.476, 85.523, 153.514, 38.085, -158.585]
  MoveL 259 to (-148.6, 230, 50) mm, rotated rx 180 ry 0 rz 90 deg; joints [-14.609, -50.999, 86.445, 155.798, 37.97, -160.49]
  MoveL 260 to (-148.6, 230, -0.5) mm, rotated rx 180 ry 0 rz 90 deg; joints [-14.609, -49.439, 86.736, 156.725, 39.666, -161.679]
  MoveL 261 to (-148.6, 230, 50) mm, rotated rx 180 ry 0 rz 90 deg; joints [-14.609, -50.999, 86.445, 155.798, 37.97, -160.49]
  MoveL 262 to (-251.4, 230, 50) mm, rotated rx 180 ry 0 rz 90 deg; joints [-11.764, -51.924, 88.066, 160.552, 37.76, -164.403]
  MoveL 263 to (-251.4, 230, -0.5) mm, rotated rx -180 ry 0 rz 90 deg; joints [-11.764, -50.339, 88.358, 161.319, 39.533, -165.384]
  MoveL 264 to (-251.4, 230, 50) mm, rotated rx 180 ry 0 rz 90 deg; joints [-11.764, -51.924, 88.066, 160.552, 37.76, -164.403]
  MoveL 265 to (-301.4, 230, 50) mm, rotated rx -180 ry 0 rz 90 deg; joints [-10.358, -52.299, 88.723, 162.89, 37.671, -166.306]
  MoveL 266 to (-301.4, 230, -0.5) mm, rotated rx -180 ry 0 rz 90 deg; joints [-10.358, -50.704, 89.015, 163.573, 39.477, -167.179]
  MoveL 267 to (-301.4, 230, 50) mm, rotated rx -180 ry 0 rz 90 deg; joints [-10.358, -52.299, 88.723, 162.89, 37.671, -166.306]
  MoveL 268 to (-351.4, 230, 50) mm, rotated rx -180 ry 0 rz 90 deg; joints [-8.939, -52.626, 89.293, 165.244, 37.592, -168.211]
  MoveL 269 to (-351.4, 230, -0.5) mm, rotated rx 180 ry 0 rz 90 deg; joints [-8.939, -51.023, 89.585, 165.839, 39.427, -168.971]
  MoveL 270 to (-351.4, 230, 50) mm, rotated rx -180 ry 0 rz 90 deg; joints [-8.939, -52.626, 89.293, 165.244, 37.592, -168.211]
  MoveL 271 to (-48.6, 420, 50) mm, rotated rx 180 ry 0 rz 90 deg; joints [-19.036, -56.892, 96.644, 151.65, 43.384, -158.588]
  MoveL 272 to (-48.6, 420, -0.5) mm, rotated rx 180 ry 0 rz 90 deg; joints [-19.036, -55.165, 96.939, 152.62, 45.171, -159.942]
  MoveL 273 to (-48.6, 420, 50) mm, rotated rx 180 ry 0 rz 90 deg; joints [-19.036, -56.892, 96.644, 151.65, 43.384, -158.588]
  MoveL 274 to (-98.6, 420, 50) mm, rotated rx 180 ry 0 rz 90 deg; joints [-17.579, -57.482, 97.646, 153.839, 43.238, -160.31]
  MoveL 275 to (-98.6, 420, -0.5) mm, rotated rx -180 ry 0 rz 90 deg; joints [-17.579, -55.736, 97.941, 154.751, 45.078, -161.581]
  MoveL 276 to (-98.6, 420, 50) mm, rotated rx 180 ry 0 rz 90 deg; joints [-17.579, -57.482, 97.646, 153.839, 43.238, -160.31]
  MoveL 277 to (-148.6, 420, 50) mm, rotated rx -180 ry 0 rz 90 deg; joints [-16.098, -58.024, 98.562, 156.057, 43.099, -162.036]
  MoveL 278 to (-148.6, 420, -0.5) mm, rotated rx 180 ry 0 rz 90 deg; joints [-16.098, -56.26, 98.859, 156.907, 44.988, -163.219]
  MoveL 279 to (-148.6, 420, 50) mm, rotated rx -180 ry 0 rz 90 deg; joints [-16.098, -58.024, 98.562, 156.057, 43.099, -162.036]
  MoveL 280 to (-251.4, 420, 50) mm, rotated rx -180 ry 0 rz 90 deg; joints [-12.985, -58.986, 100.181, 160.705, 42.842, -165.603]
  MoveL 281 to (-251.4, 420, -0.5) mm, rotated rx 180 ry 0 rz 90 deg; joints [-12.985, -57.191, 100.479, 161.413, 44.822, -166.584]
  MoveL 282 to (-251.4, 420, 50) mm, rotated rx -180 ry 0 rz 90 deg; joints [-12.985, -58.986, 100.181, 160.705, 42.842, -165.603]
  MoveL 283 to (-301.4, 420, 50) mm, rotated rx 180 ry 0 rz 90 deg; joints [-11.44, -59.379, 100.839, 163.004, 42.732, -167.346]
  MoveL 284 to (-301.4, 420, -0.5) mm, rotated rx 180 ry 0 rz 90 deg; joints [-11.44, -57.57, 101.138, 163.636, 44.752, -168.221]
  MoveL 285 to (-301.4, 420, 50) mm, rotated rx 180 ry 0 rz 90 deg; joints [-11.44, -59.379, 100.839, 163.004, 42.732, -167.346]
  MoveL 286 to (-351.4, 420, 50) mm, rotated rx 180 ry 0 rz 90 deg; joints [-9.879, -59.722, 101.411, 165.327, 42.635, -169.096]
  MoveL 287 to (-351.4, 420, -0.5) mm, rotated rx -180 ry 0 rz 90 deg; joints [-9.879, -57.902, 101.711, 165.879, 44.688, -169.86]
  MoveL 288 to (-351.4, 420, 50) mm, rotated rx 180 ry 0 rz 90 deg; joints [-9.879, -59.722, 101.411, 165.327, 42.635, -169.096]
  MoveL 289 to (-48.6, 1020, 50) mm, rotated rx -180 ry 0 rz 90 deg; joints [-27.55, -77.515, 128.518, 146.129, 56.087, -159.469]
  MoveL 290 to (-48.6, 1020, -0.5) mm, rotated rx -180 ry 0 rz 90 deg; joints [-27.55, -74.814, 128.902, 147.214, 58.665, -161.481]
  MoveL 291 to (-48.6, 1020, 50) mm, rotated rx -180 ry 0 rz 90 deg; joints [-27.55, -77.515, 128.518, 146.129, 56.087, -159.469]
  MoveL 292 to (-98.6, 1020, 50) mm, rotated rx -180 ry 0 rz 90 deg; joints [-25.595, -78.403, 129.7, 148.459, 55.673, -160.908]
  MoveL 293 to (-98.6, 1020, -0.5) mm, rotated rx 180 ry 0 rz 90 deg; joints [-25.595, -75.641, 130.092, 149.513, 58.375, -162.844]
  MoveL 294 to (-98.6, 1020, 50) mm, rotated rx -180 ry 0 rz 90 deg; joints [-25.595, -78.403, 129.7, 148.459, 55.673, -160.908]
  MoveL 295 to (-148.6, 1020, 50) mm, rotated rx 180 ry 0 rz 90 deg; joints [-23.574, -79.237, 130.795, 150.877, 55.261, -162.387]
  MoveL 296 to (-148.6, 1020, -0.5) mm, rotated rx -180 ry 0 rz 90 deg; joints [-23.574, -76.417, 131.193, 151.891, 58.087, -164.232]
  MoveL 297 to (-148.6, 1020, 50) mm, rotated rx 180 ry 0 rz 90 deg; joints [-23.574, -79.237, 130.795, 150.877, 55.261, -162.387]
  MoveL 298 to (-251.4, 1020, 50) mm, rotated rx 180 ry 0 rz 90 deg; joints [-19.22, -80.768, 132.756, 156.131, 54.444, -165.57]
  MoveL 299 to (-251.4, 1020, -0.5) mm, rotated rx 180 ry 0 rz 90 deg; joints [-19.22, -77.836, 133.168, 157.028, 57.513, -167.174]
  MoveL 300 to (-251.4, 1020, 50) mm, rotated rx 180 ry 0 rz 90 deg; joints [-19.22, -80.768, 132.756, 156.131, 54.444, -165.57]
  MoveL 301 to (-301.4, 1020, 50) mm, rotated rx 180 ry 0 rz 90 deg; joints [-17.013, -81.413, 133.564, 158.819, 54.074, -167.191]
  MoveL 302 to (-301.4, 1020, -0.5) mm, rotated rx -180 ry 0 rz 90 deg; joints [-17.013, -78.431, 133.982, 159.643, 57.253, -168.651]
  MoveL 303 to (-301.4, 1020, 50) mm, rotated rx 180 ry 0 rz 90 deg; joints [-17.013, -81.413, 133.564, 158.819, 54.074, -167.191]
  MoveL 304 to (-351.4, 1020, 50) mm, rotated rx 180 ry 0 rz 90 deg; joints [-14.752, -81.986, 134.272, 161.59, 53.732, -168.861]
  MoveL 305 to (-351.4, 1020, -0.5) mm, rotated rx 180 ry 0 rz 90 deg; joints [-14.752, -78.96, 134.696, 162.328, 57.012, -170.159]
  MoveL 306 to (-351.4, 1020, 50) mm, rotated rx 180 ry 0 rz 90 deg; joints [-14.752, -81.986, 134.272, 161.59, 53.732, -168.861]
  MoveL 307 to (-450, 50, 50) mm, rotated rx 180 ry 0 rz 90 deg; joints [-5.599, -45.905, 77.379, 169.365, 31.918, -170.944]
  MoveL 308 to (-450, 50, -0.5) mm, rotated rx -180 ry 0 rz 90 deg; joints [-5.599, -44.463, 77.676, 169.852, 33.629, -171.524]
  MoveL 309 to (-450, 50, 50) mm, rotated rx 180 ry 0 rz 90 deg; joints [-5.599, -45.905, 77.379, 169.365, 31.918, -170.944]
  MoveL 310 to (-450, 100, 50) mm, rotated rx 180 ry 0 rz 90 deg; joints [-5.732, -47.978, 81.093, 169.588, 33.552, -171.294]
  MoveL 311 to (-450, 100, -0.5) mm, rotated rx -180 ry 0 rz 90 deg; joints [-5.732, -46.49, 81.387, 170.048, 35.305, -171.851]
  MoveL 312 to (-450, 100, 50) mm, rotated rx 180 ry 0 rz 90 deg; joints [-5.732, -47.978, 81.093, 169.588, 33.552, -171.294]
  MoveL 313 to (-450, 150, 50) mm, rotated rx -180 ry 0 rz 90 deg; joints [-5.872, -49.995, 84.675, 169.755, 35.111, -171.589]
  MoveL 314 to (-450, 150, -0.5) mm, rotated rx 180 ry 0 rz 90 deg; joints [-5.872, -48.46, 84.967, 170.193, 36.911, -172.131]
  MoveL 315 to (-450, 150, 50) mm, rotated rx -180 ry 0 rz 90 deg; joints [-5.872, -49.995, 84.675, 169.755, 35.111, -171.589]
  MoveL 316 to (-450, 200, 50) mm, rotated rx -180 ry 0 rz 90 deg; joints [-6.018, -51.965, 88.139, 169.873, 36.603, -171.84]
  MoveL 317 to (-450, 200, -0.5) mm, rotated rx 180 ry 0 rz 90 deg; joints [-6.018, -50.379, 88.431, 170.294, 38.453, -172.371]
  MoveL 318 to (-450, 200, 50) mm, rotated rx -180 ry 0 rz 90 deg; joints [-6.018, -51.965, 88.139, 169.873, 36.603, -171.84]
  MoveL 319 to (-450, 250, 50) mm, rotated rx -180 ry 0 rz 90 deg; joints [-6.172, -53.895, 91.5, 169.951, 38.034, -172.054]
  MoveL 320 to (-450, 250, -0.5) mm, rotated rx -180 ry 0 rz 90 deg; joints [-6.172, -52.257, 91.792, 170.359, 39.936, -172.579]
  MoveL 321 to (-450, 250, 50) mm, rotated rx -180 ry 0 rz 90 deg; joints [-6.172, -53.895, 91.5, 169.951, 38.034, -172.054]
  MoveL 322 to (-450, 300, 50) mm, rotated rx 180 ry 0 rz 90 deg; joints [-6.334, -55.793, 94.769, 169.992, 39.406, -172.236]
  MoveL 323 to (-450, 300, -0.5) mm, rotated rx 180 ry 0 rz 90 deg; joints [-6.334, -54.1, 95.062, 170.39, 41.364, -172.758]
  MoveL 324 to (-450, 300, 50) mm, rotated rx 180 ry 0 rz 90 deg; joints [-6.334, -55.793, 94.769, 169.992, 39.406, -172.236]
  MoveL 325 to (-450, 350, 50) mm, rotated rx 180 ry 0 rz 90 deg; joints [-6.504, -57.664, 97.955, 170.001, 40.723, -172.39]
  MoveL 326 to (-450, 350, -0.5) mm, rotated rx -180 ry 0 rz 90 deg; joints [-6.504, -55.913, 98.251, 170.392, 42.741, -172.913]
  MoveL 327 to (-450, 350, 50) mm, rotated rx 180 ry 0 rz 90 deg; joints [-6.504, -57.664, 97.955, 170.001, 40.723, -172.39]
  MoveL 328 to (-450, 400, 50) mm, rotated rx -180 ry 0 rz 90 deg; joints [-6.684, -59.515, 101.065, 169.981, 41.988, -172.519]
  MoveL 329 to (-450, 400, -0.5) mm, rotated rx 180 ry 0 rz 90 deg; joints [-6.684, -57.701, 101.365, 170.367, 44.07, -173.047]
  MoveL 330 to (-450, 400, 50) mm, rotated rx -180 ry 0 rz 90 deg; joints [-6.684, -59.515, 101.065, 169.981, 41.988, -172.519]
  MoveL 331 to (-450, 450, 50) mm, rotated rx -180 ry 0 rz 90 deg; joints [-6.874, -61.35, 104.108, 169.931, 43.202, -172.625]
  MoveL 332 to (-450, 450, -0.5) mm, rotated rx -180 ry 0 rz 90 deg; joints [-6.874, -59.471, 104.412, 170.315, 45.352, -173.161]
  MoveL 333 to (-450, 450, 50) mm, rotated rx -180 ry 0 rz 90 deg; joints [-6.874, -61.35, 104.108, 169.931, 43.202, -172.625]
  MoveL 334 to (-450, 500, 50) mm, rotated rx 180 ry 0 rz 90 deg; joints [-7.075, -63.174, 107.089, 169.855, 44.366, -172.71]
  MoveL 335 to (-450, 500, -0.5) mm, rotated rx -180 ry 0 rz 90 deg; joints [-7.075, -61.226, 107.398, 170.238, 46.589, -173.257]
  MoveL 336 to (-450, 500, 50) mm, rotated rx 180 ry 0 rz 90 deg; joints [-7.075, -63.174, 107.089, 169.855, 44.366, -172.71]
  MoveL 337 to (-450, 550, 50) mm, rotated rx -180 ry 0 rz 90 deg; joints [-7.288, -64.993, 110.013, 169.751, 45.48, -172.775]
  MoveL 338 to (-450, 550, -0.5) mm, rotated rx 180 ry 0 rz 90 deg; joints [-7.288, -62.97, 110.327, 170.137, 47.782, -173.336]
  MoveL 339 to (-450, 550, 50) mm, rotated rx -180 ry 0 rz 90 deg; joints [-7.288, -64.993, 110.013, 169.751, 45.48, -172.775]
  MoveL 340 to (-450, 600, 50) mm, rotated rx 180 ry 0 rz 90 deg; joints [-7.514, -66.812, 112.884, 169.621, 46.544, -172.82]
  MoveL 341 to (-450, 600, -0.5) mm, rotated rx -180 ry 0 rz 90 deg; joints [-7.514, -64.709, 113.206, 170.011, 48.931, -173.399]
  MoveL 342 to (-450, 600, 50) mm, rotated rx 180 ry 0 rz 90 deg; joints [-7.514, -66.812, 112.884, 169.621, 46.544, -172.82]
  MoveL 343 to (-450, 650, 50) mm, rotated rx 180 ry 0 rz 90 deg; joints [-7.755, -68.635, 115.707, 169.464, 47.557, -172.846]
  MoveL 344 to (-450, 650, -0.5) mm, rotated rx -180 ry 0 rz 90 deg; joints [-7.755, -66.446, 116.036, 169.859, 50.035, -173.446]
  MoveL 345 to (-450, 650, 50) mm, rotated rx 180 ry 0 rz 90 deg; joints [-7.755, -68.635, 115.707, 169.464, 47.557, -172.846]
  MoveL 346 to (-450, 700, 50) mm, rotated rx 180 ry 0 rz 90 deg; joints [-8.012, -70.468, 118.484, 169.278, 48.517, -172.851]
  MoveL 347 to (-450, 700, -0.5) mm, rotated rx -180 ry 0 rz 90 deg; joints [-8.012, -68.187, 118.823, 169.682, 51.093, -173.477]
  MoveL 348 to (-450, 700, 50) mm, rotated rx 180 ry 0 rz 90 deg; joints [-8.012, -70.468, 118.484, 169.278, 48.517, -172.851]
  MoveL 349 to (-450, 750, 50) mm, rotated rx -180 ry 0 rz 90 deg; joints [-8.286, -72.317, 121.22, 169.063, 49.423, -172.835]
  MoveL 350 to (-450, 750, -0.5) mm, rotated rx 180 ry 0 rz 90 deg; joints [-8.286, -69.936, 121.569, 169.478, 52.105, -173.492]
  MoveL 351 to (-450, 750, 50) mm, rotated rx -180 ry 0 rz 90 deg; joints [-8.286, -72.317, 121.22, 169.063, 49.423, -172.835]
  MoveL 352 to (-450, 800, 50) mm, rotated rx 180 ry 0 rz 90 deg; joints [-8.579, -74.189, 123.917, 168.815, 50.269, -172.797]
  MoveL 353 to (-450, 800, -0.5) mm, rotated rx 180 ry 0 rz 90 deg; joints [-8.579, -71.699, 124.278, 169.244, 53.067, -173.488]
  MoveL 354 to (-450, 800, 50) mm, rotated rx 180 ry 0 rz 90 deg; joints [-8.579, -74.189, 123.917, 168.815, 50.269, -172.797]
  MoveL 355 to (-450, 850, 50) mm, rotated rx -180 ry 0 rz 90 deg; joints [-8.894, -76.089, 126.577, 168.534, 51.054, -172.734]
  MoveL 356 to (-450, 850, -0.5) mm, rotated rx 180 ry 0 rz 90 deg; joints [-8.894, -73.482, 126.951, 168.98, 53.977, -173.466]
  MoveL 357 to (-450, 850, 50) mm, rotated rx -180 ry 0 rz 90 deg; joints [-8.894, -76.089, 126.577, 168.534, 51.054, -172.734]
  MoveL 358 to (-450, 900, 50) mm, rotated rx 180 ry 0 rz 90 deg; joints [-9.232, -78.027, 129.202, 168.215, 51.77, -172.643]
  MoveL 359 to (-450, 900, -0.5) mm, rotated rx -180 ry 0 rz 90 deg; joints [-9.232, -75.292, 129.591, 168.682, 54.831, -173.424]
  MoveL 360 to (-450, 900, 50) mm, rotated rx 180 ry 0 rz 90 deg; joints [-9.232, -78.027, 129.202, 168.215, 51.77, -172.643]
  MoveL 361 to (-450, 950, 50) mm, rotated rx 180 ry 0 rz 90 deg; joints [-9.597, -80.012, 131.794, 167.855, 52.411, -172.521]
  MoveL 362 to (-450, 950, -0.5) mm, rotated rx -180 ry 0 rz 90 deg; joints [-9.597, -77.135, 132.199, 168.346, 55.622, -173.357]
  MoveL 363 to (-450, 950, 50) mm, rotated rx 180 ry 0 rz 90 deg; joints [-9.597, -80.012, 131.794, 167.855, 52.411, -172.521]
  MoveL 364 to (-450, 1000, 50) mm, rotated rx 180 ry 0 rz 90 deg; joints [-9.992, -82.053, 134.355, 167.447, 52.97, -172.363]
  MoveL 365 to (-450, 1000, -0.5) mm, rotated rx 180 ry 0 rz 90 deg; joints [-9.992, -79.022, 134.779, 167.969, 56.346, -173.264]
  MoveL 366 to (-450, 1000, 50) mm, rotated rx 180 ry 0 rz 90 deg; joints [-9.992, -82.053, 134.355, 167.447, 52.97, -172.363]
  MoveL 367 to (-450, 1050, 50) mm, rotated rx -180 ry 0 rz 90 deg; joints [-10.42, -84.166, 136.885, 166.987, 53.435, -172.161]
  MoveL 368 to (-450, 1050, -0.5) mm, rotated rx 180 ry 0 rz 90 deg; joints [-10.42, -80.963, 137.33, 167.546, 56.993, -173.14]
  MoveL 369 to (-450, 1050, 50) mm, rotated rx -180 ry 0 rz 90 deg; joints [-10.42, -84.166, 136.885, 166.987, 53.435, -172.161]
  MoveL 370 to (-450, 1100, 50) mm, rotated rx -180 ry 0 rz 90 deg; joints [-10.886, -86.364, 139.385, 166.465, 53.793, -171.907]
  MoveL 371 to (-450, 1100, -0.5) mm, rotated rx -180 ry 0 rz 90 deg; joints [-10.886, -82.972, 139.854, 167.069, 57.552, -172.977]
  MoveL 372 to (-450, 1100, 50) mm, rotated rx -180 ry 0 rz 90 deg; joints [-10.886, -86.364, 139.385, 166.465, 53.793, -171.907]
  MoveL 373 to (-450, 1150, 50) mm, rotated rx -180 ry 0 rz 90 deg; joints [-11.395, -88.668, 141.855, 165.871, 54.028, -171.589]
  MoveL 374 to (-450, 1150, -0.5) mm, rotated rx -180 ry 0 rz 90 deg; joints [-11.395, -85.064, 142.352, 166.53, 58.011, -172.768]
  MoveL 375 to (-450, 1150, 50) mm, rotated rx -180 ry 0 rz 90 deg; joints [-11.395, -88.668, 141.855, 165.871, 54.028, -171.589]
  MoveL 376 to (-450, 1200, 50) mm, rotated rx -180 ry 0 rz 90 deg; joints [-11.953, -91.1, 144.296, 165.19, 54.12, -171.192]
  MoveL 377 to (-450, 1200, -0.5) mm, rotated rx 180 ry 0 rz 90 deg; joints [-11.953, -87.26, 144.825, 165.919, 58.351, -172.502]
  MoveL 378 to (-450, 1200, 50) mm, rotated rx -180 ry 0 rz 90 deg; joints [-11.953, -91.1, 144.296, 165.19, 54.12, -171.192]
  MoveL 379 to (-450, 1250, 50) mm, rotated rx 180 ry 0 rz 90 deg; joints [-12.567, -93.692, 146.707, 164.406, 54.042, -170.693]
  MoveL 380 to (-450, 1250, -0.5) mm, rotated rx -180 ry 0 rz 90 deg; joints [-12.567, -89.587, 147.272, 165.223, 58.55, -172.164]
  MoveL 381 to (-450, 1250, 50) mm, rotated rx 180 ry 0 rz 90 deg; joints [-12.567, -93.692, 146.707, 164.406, 54.042, -170.693]
  MoveL 382 to (-450, 1300, 50) mm, rotated rx 180 ry 0 rz 90 deg; joints [-13.248, -96.482, 149.086, 163.494, 53.761, -170.064]
  MoveL 383 to (-450, 1300, -0.5) mm, rotated rx -180 ry 0 rz 90 deg; joints [-13.248, -92.077, 149.694, 164.423, 58.579, -171.731]
  MoveL 384 to (-450, 1300, 50) mm, rotated rx 180 ry 0 rz 90 deg; joints [-13.248, -96.482, 149.086, 163.494, 53.761, -170.064]
  MoveL 385 to (-450, 1350, 50) mm, rotated rx -180 ry 0 rz 90 deg; joints [-14.004, -99.519, 151.431, 162.417, 53.234, -169.26]
  MoveL 386 to (-450, 1350, -0.5) mm, rotated rx -180 ry 0 rz 90 deg; joints [-14.004, -94.776, 152.09, 163.494, 58.4, -171.174]
  MoveL 387 to (-450, 1350, 50) mm, rotated rx -180 ry 0 rz 90 deg; joints [-14.004, -99.519, 151.431, 162.417, 53.234, -169.26]
  MoveL 388 to (-450, 1400, 50) mm, rotated rx -180 ry 0 rz 90 deg; joints [-14.85, -102.871, 153.738, 161.128, 52.408, -168.221]
  MoveL 389 to (-450, 1400, -0.5) mm, rotated rx 180 ry 0 rz 90 deg; joints [-14.85, -97.745, 154.457, 162.401, 57.96, -170.448]
  MoveL 390 to (-450, 1400, 50) mm, rotated rx -180 ry 0 rz 90 deg; joints [-14.85, -102.871, 153.738, 161.128, 52.408, -168.221]
  MoveL 391 to (-450, 1450, 50) mm, rotated rx 180 ry 0 rz 70 deg; joints [-22.417, -102.648, 153.594, 130.362, 62.281, -151.309]
  MoveL 392 to (-450, 1450, -0.5) mm, rotated rx -180 ry 0 rz 70 deg; joints [-22.417, -97.548, 154.308, 132.471, 66.13, -156.151]
  MoveL 393 to (-450, 1450, 50) mm, rotated rx 180 ry 0 rz 70 deg; joints [-22.417, -102.648, 153.594, 130.362, 62.281, -151.309]
  MoveL 394 to (-578.4, 50, 50) mm, rotated rx 180 ry 0 rz 90 deg; joints [-2.182, -46.273, 78.04, 175.861, 31.835, -176.482]
  MoveL 395 to (-578.4, 50, -0.5) mm, rotated rx 180 ry 0 rz 90 deg; joints [-2.182, -44.822, 78.336, 176.053, 33.576, -176.71]
  MoveL 396 to (-578.4, 50, 50) mm, rotated rx -180 ry 0 rz 90 deg; joints [-2.182, -46.273, 78.04, 175.861, 31.835, -176.482]
  MoveL 397 to (-578.4, 100, 50) mm, rotated rx -180 ry 0 rz 90 deg; joints [-2.234, -48.344, 81.745, 175.947, 33.467, -176.617]
  MoveL 398 to (-578.4, 100, -0.5) mm, rotated rx 180 ry 0 rz 90 deg; joints [-2.234, -46.848, 82.038, 176.128, 35.252, -176.836]
  MoveL 399 to (-578.4, 100, 50) mm, rotated rx -180 ry 0 rz 90 deg; joints [-2.234, -48.344, 81.745, 175.947, 33.467, -176.617]
  MoveL 400 to (-578.4, 150, 50) mm, rotated rx 180 ry 0 rz 90 deg; joints [-2.288, -50.361, 85.32, 176.011, 35.024, -176.731]
  MoveL 401 to (-578.4, 150, -0.5) mm, rotated rx -180 ry 0 rz 90 deg; joints [-2.288, -48.816, 85.611, 176.183, 36.857, -176.944]
  MoveL 402 to (-578.4, 150, 50) mm, rotated rx 180 ry 0 rz 90 deg; joints [-2.288, -50.361, 85.32, 176.011, 35.024, -176.731]
  MoveL 403 to (-578.4, 200, 50) mm, rotated rx 180 ry 0 rz 90 deg; joints [-2.346, -52.332, 88.78, 176.056, 36.513, -176.828]
  MoveL 404 to (-578.4, 200, -0.5) mm, rotated rx 180 ry 0 rz 90 deg; joints [-2.346, -50.736, 89.071, 176.222, 38.396, -177.037]
  MoveL 405 to (-578.4, 200, 50) mm, rotated rx 180 ry 0 rz 90 deg; joints [-2.346, -52.332, 88.78, 176.056, 36.513, -176.828]
  MoveL 406 to (-578.4, 250, 50) mm, rotated rx 180 ry 0 rz 90 deg; joints [-2.406, -54.264, 92.139, 176.085, 37.939, -176.91]
  MoveL 407 to (-578.4, 250, -0.5) mm, rotated rx 180 ry 0 rz 90 deg; joints [-2.406, -52.616, 92.431, 176.246, 39.876, -177.117]
  MoveL 408 to (-578.4, 250, 50) mm, rotated rx 180 ry 0 rz 90 deg; joints [-2.406, -54.264, 92.139, 176.085, 37.939, -176.91]
  MoveL 409 to (-578.4, 300, 50) mm, rotated rx 180 ry 0 rz 90 deg; joints [-2.47, -56.166, 95.407, 176.1, 39.306, -176.98]
  MoveL 410 to (-578.4, 300, -0.5) mm, rotated rx -180 ry 0 rz 90 deg; joints [-2.47, -54.462, 95.701, 176.257, 41.3, -177.186]
  MoveL 411 to (-578.4, 300, 50) mm, rotated rx 180 ry 0 rz 90 deg; joints [-2.47, -56.166, 95.407, 176.1, 39.306, -176.98]
  MoveL 412 to (-578.4, 350, 50) mm, rotated rx 180 ry 0 rz 90 deg; joints [-2.537, -58.043, 98.594, 176.102, 40.617, -177.039]
  MoveL 413 to (-578.4, 350, -0.5) mm, rotated rx 180 ry 0 rz 90 deg; joints [-2.537, -56.279, 98.891, 176.256, 42.673, -177.246]
  MoveL 414 to (-578.4, 350, 50) mm, rotated rx 180 ry 0 rz 90 deg; joints [-2.537, -58.043, 98.594, 176.102, 40.617, -177.039]
  MoveL 415 to (-578.4, 400, 50) mm, rotated rx 180 ry 0 rz 90 deg; joints [-2.607, -59.9, 101.708, 176.092, 41.874, -177.088]
  MoveL 416 to (-578.4, 400, -0.5) mm, rotated rx -180 ry 0 rz 90 deg; joints [-2.607, -58.074, 102.009, 176.245, 43.997, -177.297]
  MoveL 417 to (-578.4, 400, 50) mm, rotated rx 180 ry 0 rz 90 deg; joints [-2.607, -59.9, 101.708, 176.092, 41.874, -177.088]
  MoveL 418 to (-578.4, 450, 50) mm, rotated rx -180 ry 0 rz 90 deg; joints [-2.682, -61.744, 104.756, 176.072, 43.079, -177.129]
  MoveL 419 to (-578.4, 450, -0.5) mm, rotated rx -180 ry 0 rz 90 deg; joints [-2.682, -59.85, 105.061, 176.224, 45.273, -177.341]
  MoveL 420 to (-578.4, 450, 50) mm, rotated rx -180 ry 0 rz 90 deg; joints [-2.682, -61.744, 104.756, 176.072, 43.079, -177.129]
  MoveL 421 to (-578.4, 500, 50) mm, rotated rx -180 ry 0 rz 90 deg; joints [-2.761, -63.578, 107.743, 176.04, 44.233, -177.161]
  MoveL 422 to (-578.4, 500, -0.5) mm, rotated rx -180 ry 0 rz 90 deg; joints [-2.761, -61.614, 108.053, 176.192, 46.502, -177.377]
  MoveL 423 to (-578.4, 500, 50) mm, rotated rx -180 ry 0 rz 90 deg; joints [-2.761, -63.578, 107.743, 176.04, 44.233, -177.161]
  MoveL 424 to (-578.4, 550, 50) mm, rotated rx -180 ry 0 rz 90 deg; joints [-2.845, -65.409, 110.674, 175.998, 45.335, -177.185]
  MoveL 425 to (-578.4, 550, -0.5) mm, rotated rx -180 ry 0 rz 90 deg; joints [-2.845, -63.368, 110.99, 176.151, 47.686, -177.407]
  MoveL 426 to (-578.4, 550, 50) mm, rotated rx -180 ry 0 rz 90 deg; joints [-2.845, -65.409, 110.674, 175.998, 45.335, -177.185]
  MoveL 427 to (-578.4, 600, 50) mm, rotated rx 180 ry 0 rz 90 deg; joints [-2.934, -67.242, 113.554, 175.946, 46.385, -177.201]
  MoveL 428 to (-578.4, 600, -0.5) mm, rotated rx 180 ry 0 rz 90 deg; joints [-2.934, -65.119, 113.878, 176.1, 48.825, -177.43]
  MoveL 429 to (-578.4, 600, 50) mm, rotated rx 180 ry 0 rz 90 deg; joints [-2.934, -67.242, 113.554, 175.946, 46.385, -177.201]
  MoveL 430 to (-578.4, 650, 50) mm, rotated rx 180 ry 0 rz 90 deg; joints [-3.029, -69.081, 116.388, 175.882, 47.381, -177.209]
  MoveL 431 to (-578.4, 650, -0.5) mm, rotated rx 180 ry 0 rz 90 deg; joints [-3.029, -66.87, 116.72, 176.04, 49.917, -177.448]
  MoveL 432 to (-578.4, 650, 50) mm, rotated rx 180 ry 0 rz 90 deg; joints [-3.029, -69.081, 116.388, 175.882, 47.381, -177.209]
  MoveL 433 to (-578.4, 700, 50) mm, rotated rx 180 ry 0 rz 90 deg; joints [-3.13, -70.933, 119.178, 175.807, 48.321, -177.209]
  MoveL 434 to (-578.4, 700, -0.5) mm, rotated rx 180 ry 0 rz 90 deg; joints [-3.13, -68.627, 119.519, 175.968, 50.961, -177.458]
  MoveL 435 to (-578.4, 700, 50) mm, rotated rx 180 ry 0 rz 90 deg; joints [-3.13, -70.933, 119.178, 175.807, 48.321, -177.209]
  MoveL 436 to (-578.4, 750, 50) mm, rotated rx 180 ry 0 rz 90 deg; joints [-3.239, -72.803, 121.927, 175.72, 49.203, -177.201]
  MoveL 437 to (-578.4, 750, -0.5) mm, rotated rx 180 ry 0 rz 90 deg; joints [-3.239, -70.395, 122.279, 175.886, 51.956, -177.462]
  MoveL 438 to (-578.4, 750, 50) mm, rotated rx 180 ry 0 rz 90 deg; joints [-3.239, -72.803, 121.927, 175.72, 49.203, -177.201]
  MoveL 439 to (-578.4, 800, 50) mm, rotated rx -180 ry 0 rz 90 deg; joints [-3.355, -74.699, 124.64, 175.62, 50.023, -177.183]
  MoveL 440 to (-578.4, 800, -0.5) mm, rotated rx 180 ry 0 rz 90 deg; joints [-3.355, -72.179, 125.004, 175.792, 52.899, -177.459]
  MoveL 441 to (-578.4, 800, 50) mm, rotated rx -180 ry 0 rz 90 deg; joints [-3.355, -74.699, 124.64, 175.62, 50.023, -177.183]
  MoveL 442 to (-578.4, 850, 50) mm, rotated rx 180 ry 0 rz 90 deg; joints [-3.48, -76.629, 127.317, 175.506, 50.775, -177.155]
  MoveL 443 to (-578.4, 850, -0.5) mm, rotated rx 180 ry 0 rz 90 deg; joints [-3.48, -73.987, 127.694, 175.686, 53.785, -177.448]
  MoveL 444 to (-578.4, 850, 50) mm, rotated rx 180 ry 0 rz 90 deg; joints [-3.48, -76.629, 127.317, 175.506, 50.775, -177.155]
  MoveL 445 to (-578.4, 900, 50) mm, rotated rx 180 ry 0 rz 90 deg; joints [-3.614, -78.6, 129.961, 175.377, 51.452, -177.115]
  MoveL 446 to (-578.4, 900, -0.5) mm, rotated rx -180 ry 0 rz 90 deg; joints [-3.614, -75.825, 130.354, 175.566, 54.61, -177.428]
  MoveL 447 to (-578.4, 900, 50) mm, rotated rx 180 ry 0 rz 90 deg; joints [-3.614, -78.6, 129.961, 175.377, 51.452, -177.115]
  MoveL 448 to (-578.4, 950, 50) mm, rotated rx -180 ry 0 rz 90 deg; joints [-3.759, -80.624, 132.574, 175.231, 52.046, -177.063]
  MoveL 449 to (-578.4, 950, -0.5) mm, rotated rx 180 ry 0 rz 90 deg; joints [-3.759, -77.702, 132.985, 175.43, 55.368, -177.399]
  MoveL 450 to (-578.4, 950, 50) mm, rotated rx -180 ry 0 rz 90 deg; joints [-3.759, -80.624, 132.574, 175.231, 52.046, -177.063]
  MoveL 451 to (-578.4, 1000, 50) mm, rotated rx -180 ry 0 rz 90 deg; joints [-3.916, -82.713, 135.158, 175.065, 52.548, -176.994]
  MoveL 452 to (-578.4, 1000, -0.5) mm, rotated rx -180 ry 0 rz 90 deg; joints [-3.916, -79.629, 135.588, 175.277, 56.049, -177.358]
  MoveL 453 to (-578.4, 1000, 50) mm, rotated rx -180 ry 0 rz 90 deg; joints [-3.916, -82.713, 135.158, 175.065, 52.548, -176.994]
  MoveL 454 to (-578.4, 1050, 50) mm, rotated rx -180 ry 0 rz 90 deg; joints [-4.087, -84.881, 137.714, 174.876, 52.943, -176.907]
  MoveL 455 to (-578.4, 1050, -0.5) mm, rotated rx 180 ry 0 rz 90 deg; joints [-4.087, -81.618, 138.166, 175.105, 56.644, -177.304]
  MoveL 456 to (-578.4, 1050, 50) mm, rotated rx -180 ry 0 rz 90 deg; joints [-4.087, -84.881, 137.714, 174.876, 52.943, -176.907]
  MoveL 457 to (-578.4, 1100, 50) mm, rotated rx 180 ry 0 rz 90 deg; joints [-4.273, -87.147, 140.242, 174.661, 53.214, -176.797]
  MoveL 458 to (-578.4, 1100, -0.5) mm, rotated rx -180 ry 0 rz 90 deg; joints [-4.273, -83.684, 140.72, 174.91, 57.139, -177.233]
  MoveL 459 to (-578.4, 1100, 50) mm, rotated rx 180 ry 0 rz 90 deg; joints [-4.273, -87.147, 140.242, 174.661, 53.214, -176.797]
  MoveL 460 to (-578.4, 1150, 50) mm, rotated rx 180 ry 0 rz 90 deg; joints [-4.478, -89.533, 142.744, 174.415, 53.341, -176.659]
  MoveL 461 to (-578.4, 1150, -0.5) mm, rotated rx -180 ry 0 rz 90 deg; joints [-4.478, -85.847, 143.251, 174.69, 57.516, -177.142]
  MoveL 462 to (-578.4, 1150, 50) mm, rotated rx 180 ry 0 rz 90 deg; joints [-4.478, -89.533, 142.744, 174.415, 53.341, -176.659]
  MoveL 463 to (-578.4, 1200, 50) mm, rotated rx 180 ry 0 rz 90 deg; joints [-4.702, -92.068, 145.219, 174.131, 53.295, -176.484]
  MoveL 464 to (-578.4, 1200, -0.5) mm, rotated rx -180 ry 0 rz 90 deg; joints [-4.702, -88.13, 145.761, 174.437, 57.753, -177.025]
  MoveL 465 to (-578.4, 1200, 50) mm, rotated rx 180 ry 0 rz 90 deg; joints [-4.702, -92.068, 145.219, 174.131, 53.295, -176.484]
  MoveL 466 to (-578.4, 1250, 50) mm, rotated rx 180 ry 0 rz 90 deg; joints [-4.951, -94.787, 147.667, 173.8, 53.041, -176.263]
  MoveL 467 to (-578.4, 1250, -0.5) mm, rotated rx -180 ry 0 rz 90 deg; joints [-4.951, -90.565, 148.248, 174.148, 57.818, -176.875]
  MoveL 468 to (-578.4, 1250, 50) mm, rotated rx 180 ry 0 rz 90 deg; joints [-4.951, -94.787, 147.667, 173.8, 53.041, -176.263]
  MoveL 469 to (-578.4, 1300, 50) mm, rotated rx 180 ry 0 rz 90 deg; joints [-5.227, -97.739, 150.087, 173.409, 52.531, -175.979]
  MoveL 470 to (-578.4, 1300, -0.5) mm, rotated rx 180 ry 0 rz 90 deg; joints [-5.227, -93.195, 150.715, 173.811, 57.672, -176.681]
  MoveL 471 to (-578.4, 1300, 50) mm, rotated rx 180 ry 0 rz 90 deg; joints [-5.227, -97.739, 150.087, 173.409, 52.531, -175.979]
  MoveL 472 to (-578.4, 1350, 50) mm, rotated rx 180 ry 0 rz 90 deg; joints [-5.535, -100.986, 152.476, 172.94, 51.702, -175.611]
  MoveL 473 to (-578.4, 1350, -0.5) mm, rotated rx -180 ry 0 rz 90 deg; joints [-5.535, -96.076, 153.16, 173.415, 57.257, -176.427]
  MoveL 474 to (-578.4, 1350, 50) mm, rotated rx 180 ry 0 rz 90 deg; joints [-5.535, -100.986, 152.476, 172.94, 51.702, -175.611]
  MoveL 475 to (-578.4, 1400, 50) mm, rotated rx 180 ry 0 rz 90 deg; joints [-5.882, -104.615, 154.831, 172.364, 50.467, -175.122]
  MoveL 476 to (-578.4, 1400, -0.5) mm, rotated rx -180 ry 0 rz 70 deg; joints [-12.877, -96.991, 153.881, 142.344, 62.693, -160.506]
  MoveL 477 to (-578.4, 1400, 50) mm, rotated rx 180 ry 0 rz 90 deg; joints [-5.882, -104.615, 154.831, 172.364, 50.467, -175.122]
  MoveL 478 to (-578.4, 1450, 50) mm, rotated rx -180 ry 0 rz 50 deg; joints [-18.777, -100.129, 151.872, 115.454, 71.278, -146.007]
  MoveL 479 to (-578.4, 1450, -0.5) mm, rotated rx 180 ry 0 rz 50 deg; joints [-18.777, -95.317, 152.541, 117.006, 73.703, -151.163]
  MoveL 480 to (-578.4, 1450, 50) mm, rotated rx -180 ry 0 rz 50 deg; joints [-18.777, -100.129, 151.872, 115.454, 71.278, -146.007]
  MoveL 481 to (-514.2, 300, 50) mm, rotated rx -180 ry 0 rz 90 deg; joints [-4.407, -56.021, 95.158, 173.039, 39.345, -174.606]
  MoveL 482 to (-514.2, 300, -0.5) mm, rotated rx -180 ry 0 rz 90 deg; joints [-4.407, -54.32, 95.452, 173.318, 41.325, -174.972]
  MoveL 483 to (-514.2, 300, 50) mm, rotated rx -180 ry 0 rz 90 deg; joints [-4.407, -56.021, 95.158, 173.039, 39.345, -174.606]
  MoveL 484 to (-514.2, 650, 50) mm, rotated rx -180 ry 0 rz 90 deg; joints [-5.401, -68.907, 116.122, 172.659, 47.45, -175.021]
  MoveL 485 to (-514.2, 650, -0.5) mm, rotated rx 180 ry 0 rz 90 deg; joints [-5.401, -66.704, 116.453, 172.938, 49.963, -175.444]
  MoveL 486 to (-514.2, 650, 50) mm, rotated rx -180 ry 0 rz 90 deg; joints [-5.401, -68.907, 116.122, 172.659, 47.45, -175.021]
  MoveL 487 to (-476, 1150, 50) mm, rotated rx -180 ry 0 rz 90 deg; joints [-10.014, -88.901, 142.097, 167.563, 53.846, -172.587]
  MoveL 488 to (-476, 1150, -0.5) mm, rotated rx -180 ry 0 rz 90 deg; joints [-10.014, -85.275, 142.597, 168.152, 57.88, -173.635]
  MoveL 489 to (-476, 1150, 50) mm, rotated rx -180 ry 0 rz 90 deg; joints [-10.014, -88.901, 142.097, 167.563, 53.846, -172.587]
  MoveL 490 to (-514.2, 1150, 50) mm, rotated rx 180 ry 0 rz 90 deg; joints [-7.965, -89.192, 142.396, 170.088, 53.616, -174.082]
  MoveL 491 to (-514.2, 1150, -0.5) mm, rotated rx 180 ry 0 rz 90 deg; joints [-7.965, -85.538, 142.899, 170.566, 57.714, -174.928]
  MoveL 492 to (-514.2, 1150, 50) mm, rotated rx 180 ry 0 rz 90 deg; joints [-7.965, -89.192, 142.396, 170.088, 53.616, -174.082]
  MoveL 493 to (-552.4, 1150, 50) mm, rotated rx -180 ry 0 rz 90 deg; joints [-5.896, -89.418, 142.626, 172.652, 53.435, -175.607]
  MoveL 494 to (-552.4, 1150, -0.5) mm, rotated rx 180 ry 0 rz 90 deg; joints [-5.896, -85.742, 143.132, 173.011, 57.584, -176.24]
  MoveL 495 to (-552.4, 1150, 50) mm, rotated rx -180 ry 0 rz 90 deg; joints [-5.896, -89.418, 142.626, 172.652, 53.435, -175.607]
  MoveL 496 to (-655, 50, 50) mm, rotated rx -180 ry 0 rz 90 deg; joints [-0.134, -46.338, 78.157, 179.746, 31.82, -179.784]
  MoveL 497 to (-655, 50, -0.5) mm, rotated rx 180 ry 0 rz 90 deg; joints [-0.134, -44.886, 78.453, 179.758, 33.567, -179.798]
  MoveL 498 to (-655, 50, 50) mm, rotated rx -180 ry 0 rz 90 deg; joints [-0.134, -46.338, 78.157, 179.746, 31.82, -179.784]
  MoveL 499 to (-655, 100, 50) mm, rotated rx 180 ry 0 rz 90 deg; joints [-0.137, -48.409, 81.86, 179.752, 33.452, -179.793]
  MoveL 500 to (-655, 100, -0.5) mm, rotated rx -180 ry 0 rz 90 deg; joints [-0.137, -46.911, 82.153, 179.763, 35.243, -179.806]
  MoveL 501 to (-655, 100, 50) mm, rotated rx 180 ry 0 rz 90 deg; joints [-0.137, -48.409, 81.86, 179.752, 33.452, -179.793]
  MoveL 502 to (-655, 150, 50) mm, rotated rx -180 ry 0 rz 90 deg; joints [-0.14, -50.425, 85.434, 179.755, 35.009, -179.8]
  MoveL 503 to (-655, 150, -0.5) mm, rotated rx 180 ry 0 rz 90 deg; joints [-0.14, -48.879, 85.726, 179.766, 36.847, -179.813]
  MoveL 504 to (-655, 150, 50) mm, rotated rx -180 ry 0 rz 90 deg; joints [-0.14, -50.425, 85.434, 179.755, 35.009, -179.8]
  MoveL 505 to (-655, 200, 50) mm, rotated rx 180 ry 0 rz 90 deg; joints [-0.144, -52.397, 88.893, 179.758, 36.497, -179.806]
  MoveL 506 to (-655, 200, -0.5) mm, rotated rx -180 ry 0 rz 90 deg; joints [-0.144, -50.799, 89.185, 179.768, 38.386, -179.818]
  MoveL 507 to (-655, 200, 50) mm, rotated rx 180 ry 0 rz 90 deg; joints [-0.144, -52.397, 88.893, 179.758, 36.497, -179.806]
  MoveL 508 to (-655, 250, 50) mm, rotated rx 180 ry 0 rz 90 deg; joints [-0.148, -54.33, 92.252, 179.76, 37.922, -179.811]
  MoveL 509 to (-655, 250, -0.5) mm, rotated rx 180 ry 0 rz 90 deg; joints [-0.148, -52.679, 92.544, 179.77, 39.865, -179.823]
  MoveL 510 to (-655, 250, 50) mm, rotated rx 180 ry 0 rz 90 deg; joints [-0.148, -54.33, 92.252, 179.76, 37.922, -179.811]
  MoveL 511 to (-655, 300, 50) mm, rotated rx -180 ry 0 rz 90 deg; joints [-0.151, -56.232, 95.52, 179.761, 39.288, -179.815]
  MoveL 512 to (-655, 300, -0.5) mm, rotated rx 180 ry 0 rz 90 deg; joints [-0.151, -54.526, 95.814, 179.771, 41.289, -179.828]
  MoveL 513 to (-655, 300, 50) mm, rotated rx -180 ry 0 rz 90 deg; joints [-0.151, -56.232, 95.52, 179.761, 39.288, -179.815]
  MoveL 514 to (-655, 350, 50) mm, rotated rx 180 ry 0 rz 90 deg; joints [-0.156, -58.11, 98.708, 179.761, 40.598, -179.819]
  MoveL 515 to (-655, 350, -0.5) mm, rotated rx 180 ry 0 rz 90 deg; joints [-0.156, -56.344, 99.005, 179.77, 42.661, -179.831]
  MoveL 516 to (-655, 350, 50) mm, rotated rx 180 ry 0 rz 90 deg; joints [-0.156, -58.11, 98.708, 179.761, 40.598, -179.819]
  MoveL 517 to (-655, 400, 50) mm, rotated rx 180 ry 0 rz 90 deg; joints [-0.16, -59.969, 101.822, 179.76, 41.854, -179.822]
  MoveL 518 to (-655, 400, -0.5) mm, rotated rx -180 ry 0 rz 90 deg; joints [-0.16, -58.14, 102.123, 179.77, 43.983, -179.834]
  MoveL 519 to (-655, 400, 50) mm, rotated rx 180 ry 0 rz 90 deg; joints [-0.16, -59.969, 101.822, 179.76, 41.854, -179.822]
  MoveL 520 to (-655, 450, 50) mm, rotated rx 180 ry 0 rz 90 deg; joints [-0.164, -61.814, 104.871, 179.759, 43.057, -179.824]
  MoveL 521 to (-655, 450, -0.5) mm, rotated rx -180 ry 0 rz 90 deg; joints [-0.164, -59.918, 105.176, 179.768, 45.258, -179.837]
  MoveL 522 to (-655, 450, 50) mm, rotated rx 180 ry 0 rz 90 deg; joints [-0.164, -61.814, 104.871, 179.759, 43.057, -179.824]
  MoveL 523 to (-655, 500, 50) mm, rotated rx 180 ry 0 rz 90 deg; joints [-0.169, -63.65, 107.859, 179.757, 44.209, -179.826]
  MoveL 524 to (-655, 500, -0.5) mm, rotated rx -180 ry 0 rz 90 deg; joints [-0.169, -61.683, 108.169, 179.767, 46.487, -179.839]
  MoveL 525 to (-655, 500, 50) mm, rotated rx 180 ry 0 rz 90 deg; joints [-0.169, -63.65, 107.859, 179.757, 44.209, -179.826]
  MoveL 526 to (-655, 550, 50) mm, rotated rx 180 ry 0 rz 90 deg; joints [-0.174, -65.483, 110.791, 179.755, 45.309, -179.827]
  MoveL 527 to (-655, 550, -0.5) mm, rotated rx 180 ry 0 rz 90 deg; joints [-0.174, -63.439, 111.108, 179.764, 47.669, -179.841]
  MoveL 528 to (-655, 550, 50) mm, rotated rx 180 ry 0 rz 90 deg; joints [-0.174, -65.483, 110.791, 179.755, 45.309, -179.827]
  MoveL 529 to (-655, 600, 50) mm, rotated rx -180 ry 0 rz 90 deg; joints [-0.18, -67.318, 113.673, 179.751, 46.356, -179.828]
  MoveL 530 to (-655, 600, -0.5) mm, rotated rx 180 ry 0 rz 90 deg; joints [-0.18, -65.192, 113.997, 179.761, 48.806, -179.842]
  MoveL 531 to (-655, 600, 50) mm, rotated rx -180 ry 0 rz 90 deg; joints [-0.18, -67.318, 113.673, 179.751, 46.356, -179.828]
  MoveL 532 to (-655, 650, 50) mm, rotated rx 180 ry 0 rz 90 deg; joints [-0.186, -69.16, 116.509, 179.747, 47.349, -179.829]
  MoveL 533 to (-655, 650, -0.5) mm, rotated rx 180 ry 0 rz 90 deg; joints [-0.186, -66.946, 116.841, 179.757, 49.896, -179.844]
  MoveL 534 to (-655, 650, 50) mm, rotated rx 180 ry 0 rz 90 deg; joints [-0.186, -69.16, 116.509, 179.747, 47.349, -179.829]
  MoveL 535 to (-655, 700, 50) mm, rotated rx 180 ry 0 rz 90 deg; joints [-0.192, -71.015, 119.301, 179.743, 48.286, -179.829]
  MoveL 536 to (-655, 700, -0.5) mm, rotated rx -180 ry 0 rz 90 deg; joints [-0.192, -68.705, 119.643, 179.753, 50.938, -179.844]
  MoveL 537 to (-655, 700, 50) mm, rotated rx 180 ry 0 rz 90 deg; joints [-0.192, -71.015, 119.301, 179.743, 48.286, -179.829]
  MoveL 538 to (-655, 750, 50) mm, rotated rx 180 ry 0 rz 90 deg; joints [-0.199, -72.89, 122.053, 179.737, 49.164, -179.828]
  MoveL 539 to (-655, 750, -0.5) mm, rotated rx 180 ry 0 rz 90 deg; joints [-0.199, -70.476, 122.406, 179.748, 51.929, -179.844]
  MoveL 540 to (-655, 750, 50) mm, rotated rx 180 ry 0 rz 90 deg; joints [-0.199, -72.89, 122.053, 179.737, 49.164, -179.828]
  MoveL 541 to (-655, 800, 50) mm, rotated rx -180 ry 0 rz 90 deg; joints [-0.206, -74.79, 124.768, 179.731, 49.978, -179.827]
  MoveL 542 to (-655, 800, -0.5) mm, rotated rx -180 ry 0 rz 90 deg; joints [-0.206, -72.265, 125.133, 179.742, 52.868, -179.844]
  MoveL 543 to (-655, 800, 50) mm, rotated rx -180 ry 0 rz 90 deg; joints [-0.206, -74.79, 124.768, 179.731, 49.978, -179.827]
  MoveL 544 to (-655, 850, 50) mm, rotated rx -180 ry 0 rz 90 deg; joints [-0.213, -76.725, 127.448, 179.724, 50.724, -179.825]
  MoveL 545 to (-655, 850, -0.5) mm, rotated rx -180 ry 0 rz 90 deg; joints [-0.213, -74.077, 127.827, 179.735, 53.75, -179.843]
  MoveL 546 to (-655, 850, 50) mm, rotated rx -180 ry 0 rz 90 deg; joints [-0.213, -76.725, 127.448, 179.724, 50.724, -179.825]
  MoveL 547 to (-655, 900, 50) mm, rotated rx -180 ry 0 rz 90 deg; joints [-0.222, -78.703, 130.096, 179.716, 51.394, -179.823]
  MoveL 548 to (-655, 900, -0.5) mm, rotated rx 180 ry 0 rz 90 deg; joints [-0.222, -75.92, 130.49, 179.728, 54.57, -179.842]
  MoveL 549 to (-655, 900, 50) mm, rotated rx -180 ry 0 rz 90 deg; joints [-0.222, -78.703, 130.096, 179.716, 51.394, -179.823]
  MoveL 550 to (-655, 950, 50) mm, rotated rx 180 ry 0 rz 90 deg; joints [-0.231, -80.734, 132.713, 179.707, 51.979, -179.82]
  MoveL 551 to (-655, 950, -0.5) mm, rotated rx 180 ry 0 rz 90 deg; joints [-0.231, -77.804, 133.125, 179.72, 55.321, -179.84]
  MoveL 552 to (-655, 950, 50) mm, rotated rx 180 ry 0 rz 90 deg; joints [-0.231, -80.734, 132.713, 179.707, 51.979, -179.82]
  MoveL 553 to (-655, 1000, 50) mm, rotated rx -180 ry 0 rz 90 deg; joints [-0.24, -82.832, 135.301, 179.697, 52.47, -179.815]
  MoveL 554 to (-655, 1000, -0.5) mm, rotated rx 180 ry 0 rz 90 deg; joints [-0.24, -79.738, 135.732, 179.71, 55.994, -179.838]
  MoveL 555 to (-655, 1000, 50) mm, rotated rx -180 ry 0 rz 90 deg; joints [-0.24, -82.832, 135.301, 179.697, 52.47, -179.815]
  MoveL 556 to (-655, 1050, 50) mm, rotated rx 180 ry 0 rz 90 deg; joints [-0.251, -85.01, 137.861, 179.685, 52.851, -179.81]
  MoveL 557 to (-655, 1050, -0.5) mm, rotated rx -180 ry 0 rz 90 deg; joints [-0.251, -81.736, 138.315, 179.699, 56.58, -179.834]
  MoveL 558 to (-655, 1050, 50) mm, rotated rx 180 ry 0 rz 90 deg; joints [-0.251, -85.01, 137.861, 179.685, 52.851, -179.81]
  MoveL 559 to (-655, 1100, 50) mm, rotated rx 180 ry 0 rz 90 deg; joints [-0.262, -87.289, 140.395, 179.672, 53.107, -179.803]
  MoveL 560 to (-655, 1100, -0.5) mm, rotated rx 180 ry 0 rz 90 deg; joints [-0.262, -83.813, 140.875, 179.687, 57.062, -179.83]
  MoveL 561 to (-655, 1100, 50) mm, rotated rx 180 ry 0 rz 90 deg; joints [-0.262, -87.289, 140.395, 179.672, 53.107, -179.803]
  MoveL 562 to (-655, 1150, 50) mm, rotated rx 180 ry 0 rz 90 deg; joints [-0.275, -89.69, 142.902, 179.657, 53.213, -179.794]
  MoveL 563 to (-655, 1150, -0.5) mm, rotated rx -180 ry 0 rz 90 deg; joints [-0.275, -85.989, 143.412, 179.674, 57.424, -179.824]
  MoveL 564 to (-655, 1150, 50) mm, rotated rx 180 ry 0 rz 90 deg; joints [-0.275, -89.69, 142.902, 179.657, 53.213, -179.794]
  MoveL 565 to (-655, 1200, 50) mm, rotated rx -180 ry 0 rz 90 deg; joints [-0.289, -92.243, 145.383, 179.639, 53.141, -179.783]
  MoveL 566 to (-655, 1200, -0.5) mm, rotated rx 180 ry 0 rz 90 deg; joints [-0.289, -88.288, 145.928, 179.658, 57.64, -179.817]
  MoveL 567 to (-655, 1200, 50) mm, rotated rx -180 ry 0 rz 90 deg; joints [-0.289, -92.243, 145.383, 179.639, 53.141, -179.783]
  MoveL 568 to (-655, 1250, 50) mm, rotated rx -180 ry 0 rz 90 deg; joints [-0.304, -94.987, 147.838, 179.618, 52.852, -179.77]
  MoveL 569 to (-655, 1250, -0.5) mm, rotated rx -180 ry 0 rz 90 deg; joints [-0.304, -90.744, 148.423, 179.64, 57.68, -179.808]
  MoveL 570 to (-655, 1250, 50) mm, rotated rx -180 ry 0 rz 90 deg; joints [-0.304, -94.987, 147.838, 179.618, 52.852, -179.77]
  MoveL 571 to (-783.4, 50, 50) mm, rotated rx 180 ry 0 rz 90 deg; joints [3.297, -46.188, 77.889, 186.256, 31.854, -185.32]
  MoveL 572 to (-783.4, 50, -0.5) mm, rotated rx 180 ry 0 rz 90 deg; joints [3.297, -44.74, 78.185, 185.967, 33.588, -184.977]
  MoveL 573 to (-783.4, 50, 50) mm, rotated rx 180 ry 0 rz 90 deg; joints [3.297, -46.188, 77.889, 186.256, 31.854, -185.32]
  MoveL 574 to (-783.4, 100, 50) mm, rotated rx -180 ry 0 rz 90 deg; joints [3.376, -48.26, 81.596, 186.127, 33.486, -185.116]
  MoveL 575 to (-783.4, 100, -0.5) mm, rotated rx 180 ry 0 rz 90 deg; joints [3.376, -46.766, 81.889, 185.854, 35.265, -184.785]
  MoveL 576 to (-783.4, 100, 50) mm, rotated rx -180 ry 0 rz 90 deg; joints [3.376, -48.26, 81.596, 186.127, 33.486, -185.116]
  MoveL 577 to (-783.4, 150, 50) mm, rotated rx 180 ry 0 rz 90 deg; joints [3.458, -50.277, 85.172, 186.03, 35.044, -184.943]
  MoveL 578 to (-783.4, 150, -0.5) mm, rotated rx 180 ry 0 rz 90 deg; joints [3.458, -48.734, 85.464, 185.77, 36.869, -184.622]
  MoveL 579 to (-783.4, 150, 50) mm, rotated rx 180 ry 0 rz 90 deg; joints [3.458, -50.277, 85.172, 186.03, 35.044, -184.943]
  MoveL 580 to (-783.4, 200, 50) mm, rotated rx 180 ry 0 rz 90 deg; joints [3.545, -52.248, 88.633, 185.962, 36.534, -184.796]
  MoveL 581 to (-783.4, 200, -0.5) mm, rotated rx -180 ry 0 rz 90 deg; joints [3.545, -50.654, 88.925, 185.712, 38.409, -184.481]
  MoveL 582 to (-783.4, 200, 50) mm, rotated rx 180 ry 0 rz 90 deg; joints [3.545, -52.248, 88.633, 185.962, 36.534, -184.796]
  MoveL 583 to (-783.4, 250, 50) mm, rotated rx -180 ry 0 rz 90 deg; joints [3.636, -54.18, 91.992, 185.917, 37.961, -184.672]
  MoveL 584 to (-783.4, 250, -0.5) mm, rotated rx -180 ry 0 rz 90 deg; joints [3.636, -52.534, 92.285, 185.675, 39.89, -184.36]
  MoveL 585 to (-783.4, 250, 50) mm, rotated rx -180 ry 0 rz 90 deg; joints [3.636, -54.18, 91.992, 185.917, 37.961, -184.672]
  MoveL 586 to (-783.4, 300, 50) mm, rotated rx 180 ry 0 rz 90 deg; joints [3.732, -56.081, 95.261, 185.894, 39.329, -184.566]
  MoveL 587 to (-783.4, 300, -0.5) mm, rotated rx -180 ry 0 rz 90 deg; joints [3.732, -54.379, 95.555, 185.658, 41.315, -184.255]
  MoveL 588 to (-783.4, 300, 50) mm, rotated rx 180 ry 0 rz 90 deg; joints [3.732, -56.081, 95.261, 185.894, 39.329, -184.566]
  MoveL 589 to (-783.4, 350, 50) mm, rotated rx 180 ry 0 rz 90 deg; joints [3.833, -57.956, 98.448, 185.89, 40.642, -184.476]
  MoveL 590 to (-783.4, 350, -0.5) mm, rotated rx 180 ry 0 rz 90 deg; joints [3.833, -56.195, 98.745, 185.658, 42.689, -184.165]
  MoveL 591 to (-783.4, 350, 50) mm, rotated rx 180 ry 0 rz 90 deg; joints [3.833, -57.956, 98.448, 185.89, 40.642, -184.476]
  MoveL 592 to (-783.4, 400, 50) mm, rotated rx -180 ry 0 rz 90 deg; joints [3.939, -59.812, 101.561, 185.904, 41.901, -184.402]
  MoveL 593 to (-783.4, 400, -0.5) mm, rotated rx -180 ry 0 rz 90 deg; joints [3.939, -57.988, 101.861, 185.674, 44.014, -184.087]
  MoveL 594 to (-783.4, 400, 50) mm, rotated rx -180 ry 0 rz 90 deg; joints [3.939, -59.812, 101.561, 185.904, 41.901, -184.402]
  MoveL 595 to (-783.4, 450, 50) mm, rotated rx 180 ry 0 rz 90 deg; joints [4.052, -61.653, 104.608, 185.935, 43.108, -184.34]
  MoveL 596 to (-783.4, 450, -0.5) mm, rotated rx 180 ry 0 rz 90 deg; joints [4.052, -59.763, 104.912, 185.706, 45.291, -184.021]
  MoveL 597 to (-783.4, 450, 50) mm, rotated rx 180 ry 0 rz 90 deg; joints [4.052, -61.653, 104.608, 185.935, 43.108, -184.34]
  MoveL 598 to (-783.4, 500, 50) mm, rotated rx 180 ry 0 rz 90 deg; joints [4.171, -63.486, 107.593, 185.982, 44.264, -184.291]
  MoveL 599 to (-783.4, 500, -0.5) mm, rotated rx -180 ry 0 rz 90 deg; joints [4.171, -61.525, 107.903, 185.753, 46.523, -183.965]
  MoveL 600 to (-783.4, 500, 50) mm, rotated rx 180 ry 0 rz 90 deg; joints [4.171, -63.486, 107.593, 185.982, 44.264, -184.291]
  MoveL 601 to (-783.4, 550, 50) mm, rotated rx -180 ry 0 rz 90 deg; joints [4.298, -65.314, 110.523, 186.045, 45.368, -184.255]
  MoveL 602 to (-783.4, 550, -0.5) mm, rotated rx 180 ry 0 rz 90 deg; joints [4.298, -63.277, 110.838, 185.815, 47.709, -183.92]
  MoveL 603 to (-783.4, 550, 50) mm, rotated rx -180 ry 0 rz 90 deg; joints [4.298, -65.314, 110.523, 186.045, 45.368, -184.255]
  MoveL 604 to (-783.4, 600, 50) mm, rotated rx -180 ry 0 rz 90 deg; joints [4.432, -67.143, 113.401, 186.124, 46.422, -184.23]
  MoveL 605 to (-783.4, 600, -0.5) mm, rotated rx -180 ry 0 rz 90 deg; joints [4.432, -65.025, 113.724, 185.891, 48.849, -183.884]
  MoveL 606 to (-783.4, 600, 50) mm, rotated rx -180 ry 0 rz 90 deg; joints [4.432, -67.143, 113.401, 186.124, 46.422, -184.23]
  MoveL 607 to (-783.4, 650, 50) mm, rotated rx -180 ry 0 rz 90 deg; joints [4.575, -68.978, 116.232, 186.219, 47.422, -184.217]
  MoveL 608 to (-783.4, 650, -0.5) mm, rotated rx -180 ry 0 rz 90 deg; joints [4.575, -66.773, 116.563, 185.982, 49.944, -183.858]
  MoveL 609 to (-783.4, 650, 50) mm, rotated rx -180 ry 0 rz 90 deg; joints [4.575, -68.978, 116.232, 186.219, 47.422, -184.217]
  MoveL 610 to (-783.4, 700, 50) mm, rotated rx -180 ry 0 rz 90 deg; joints [4.728, -70.826, 119.019, 186.332, 48.367, -184.216]
  MoveL 611 to (-783.4, 700, -0.5) mm, rotated rx -180 ry 0 rz 90 deg; joints [4.728, -68.526, 119.359, 186.089, 50.992, -183.841]
  MoveL 612 to (-783.4, 700, 50) mm, rotated rx -180 ry 0 rz 90 deg; joints [4.728, -70.826, 119.019, 186.332, 48.367, -184.216]
  MoveL 613 to (-783.4, 750, 50) mm, rotated rx -180 ry 0 rz 90 deg; joints [4.891, -72.691, 121.765, 186.462, 49.254, -184.228]
  MoveL 614 to (-783.4, 750, -0.5) mm, rotated rx 180 ry 0 rz 90 deg; joints [4.891, -70.289, 122.117, 186.212, 51.991, -183.835]
  MoveL 615 to (-783.4, 750, 50) mm, rotated rx -180 ry 0 rz 90 deg; joints [4.891, -72.691, 121.765, 186.462, 49.254, -184.228]
  MoveL 616 to (-783.4, 800, 50) mm, rotated rx -180 ry 0 rz 90 deg; joints [5.066, -74.582, 124.474, 186.611, 50.08, -184.254]
  MoveL 617 to (-783.4, 800, -0.5) mm, rotated rx 180 ry 0 rz 90 deg; joints [5.066, -72.069, 124.837, 186.353, 52.938, -183.839]
  MoveL 618 to (-783.4, 800, 50) mm, rotated rx -180 ry 0 rz 90 deg; joints [5.066, -74.582, 124.474, 186.611, 50.08, -184.254]
  MoveL 619 to (-783.4, 850, 50) mm, rotated rx 180 ry 0 rz 90 deg; joints [5.254, -76.504, 127.147, 186.782, 50.84, -184.295]
  MoveL 620 to (-783.4, 850, -0.5) mm, rotated rx -180 ry 0 rz 90 deg; joints [5.254, -73.871, 127.524, 186.513, 53.83, -183.855]
  MoveL 621 to (-783.4, 850, 50) mm, rotated rx 180 ry 0 rz 90 deg; joints [5.254, -76.504, 127.147, 186.782, 50.84, -184.295]
  MoveL 622 to (-783.4, 900, 50) mm, rotated rx -180 ry 0 rz 90 deg; joints [5.456, -78.468, 129.787, 186.975, 51.526, -184.353]
  MoveL 623 to (-783.4, 900, -0.5) mm, rotated rx 180 ry 0 rz 90 deg; joints [5.456, -75.702, 130.179, 186.693, 54.662, -183.883]
  MoveL 624 to (-783.4, 900, 50) mm, rotated rx -180 ry 0 rz 90 deg; joints [5.456, -78.468, 129.787, 186.975, 51.526, -184.353]
  MoveL 625 to (-783.4, 950, 50) mm, rotated rx -180 ry 0 rz 90 deg; joints [5.674, -80.483, 132.395, 187.195, 52.132, -184.431]
  MoveL 626 to (-783.4, 950, -0.5) mm, rotated rx 180 ry 0 rz 90 deg; joints [5.674, -77.572, 132.804, 186.896, 55.427, -183.926]
  MoveL 627 to (-783.4, 950, 50) mm, rotated rx -180 ry 0 rz 90 deg; joints [5.674, -80.483, 132.395, 187.195, 52.132, -184.431]
  MoveL 628 to (-783.4, 1000, 50) mm, rotated rx -180 ry 0 rz 90 deg; joints [5.91, -82.561, 134.973, 187.443, 52.647, -184.532]
  MoveL 629 to (-783.4, 1000, -0.5) mm, rotated rx 180 ry 0 rz 90 deg; joints [5.91, -79.489, 135.402, 187.125, 56.119, -183.986]
  MoveL 630 to (-783.4, 1000, 50) mm, rotated rx -180 ry 0 rz 90 deg; joints [5.91, -82.561, 134.973, 187.443, 52.647, -184.532]
  MoveL 631 to (-783.4, 1050, 50) mm, rotated rx 180 ry 0 rz 90 deg; joints [6.167, -84.716, 137.523, 187.725, 53.058, -184.661]
  MoveL 632 to (-783.4, 1050, -0.5) mm, rotated rx 180 ry 0 rz 90 deg; joints [6.167, -81.467, 137.974, 187.383, 56.726, -184.066]
  MoveL 633 to (-783.4, 1050, 50) mm, rotated rx 180 ry 0 rz 90 deg; joints [6.167, -84.716, 137.523, 187.725, 53.058, -184.661]
  MoveL 634 to (-783.4, 1100, 50) mm, rotated rx -180 ry 0 rz 90 deg; joints [6.447, -86.966, 140.045, 188.045, 53.351, -184.823]
  MoveL 635 to (-783.4, 1100, -0.5) mm, rotated rx 180 ry 0 rz 90 deg; joints [6.447, -83.519, 140.521, 187.674, 57.237, -184.17]
  MoveL 636 to (-783.4, 1100, 50) mm, rotated rx -180 ry 0 rz 90 deg; joints [6.447, -86.966, 140.045, 188.045, 53.351, -184.823]
  MoveL 637 to (-783.4, 1150, 50) mm, rotated rx -180 ry 0 rz 90 deg; joints [6.754, -89.332, 142.539, 188.412, 53.504, -185.027]
  MoveL 638 to (-783.4, 1150, -0.5) mm, rotated rx -180 ry 0 rz 90 deg; joints [6.754, -85.665, 143.044, 188.004, 57.633, -184.305]
  MoveL 639 to (-783.4, 1150, 50) mm, rotated rx -180 ry 0 rz 90 deg; joints [6.754, -89.332, 142.539, 188.412, 53.504, -185.027]
  MoveL 640 to (-783.4, 1200, 50) mm, rotated rx 180 ry 0 rz 90 deg; joints [7.091, -91.842, 145.006, 188.835, 53.491, -185.283]
  MoveL 641 to (-783.4, 1200, -0.5) mm, rotated rx -180 ry 0 rz 90 deg; joints [7.091, -87.928, 145.545, 188.38, 57.895, -184.476]
  MoveL 642 to (-783.4, 1200, 50) mm, rotated rx 180 ry 0 rz 90 deg; joints [7.091, -91.842, 145.006, 188.835, 53.491, -185.283]
  MoveL 643 to (-783.4, 1250, 50) mm, rotated rx -180 ry 0 rz 90 deg; joints [7.463, -94.531, 147.446, 189.325, 53.28, -185.607]
  MoveL 644 to (-783.4, 1250, -0.5) mm, rotated rx 180 ry 0 rz 90 deg; joints [7.463, -90.337, 148.023, 188.811, 57.993, -184.697]
  MoveL 645 to (-783.4, 1250, 50) mm, rotated rx -180 ry 0 rz 90 deg; joints [7.463, -94.531, 147.446, 189.325, 53.28, -185.607]
  MoveL 646 to (-681, 1150, 50) mm, rotated rx 180 ry 0 rz 90 deg; joints [1.155, -89.68, 142.892, 181.442, 53.221, -180.863]
  MoveL 647 to (-681, 1150, -0.5) mm, rotated rx 180 ry 0 rz 90 deg; joints [1.155, -85.98, 143.402, 181.37, 57.43, -180.738]
  MoveL 648 to (-681, 1150, 50) mm, rotated rx 180 ry 0 rz 90 deg; joints [1.155, -89.68, 142.892, 181.442, 53.221, -180.863]
  MoveL 649 to (-719.2, 1150, 50) mm, rotated rx -180 ry 0 rz 90 deg; joints [3.252, -89.608, 142.819, 184.058, 53.28, -182.429]
  MoveL 650 to (-719.2, 1150, -0.5) mm, rotated rx 180 ry 0 rz 90 deg; joints [3.252, -85.914, 143.328, 183.858, 57.472, -182.076]
  MoveL 651 to (-719.2, 1150, 50) mm, rotated rx -180 ry 0 rz 90 deg; joints [3.252, -89.608, 142.819, 184.058, 53.28, -182.429]
  MoveL 652 to (-757.4, 1150, 50) mm, rotated rx -180 ry 0 rz 90 deg; joints [5.34, -89.467, 142.676, 186.658, 53.395, -183.981]
  MoveL 653 to (-757.4, 1150, -0.5) mm, rotated rx -180 ry 0 rz 90 deg; joints [5.34, -85.787, 143.183, 186.332, 57.555, -183.407]
  MoveL 654 to (-757.4, 1150, 50) mm, rotated rx -180 ry 0 rz 90 deg; joints [5.34, -89.467, 142.676, 186.658, 53.395, -183.981]
  MoveL 655 to (-890, 50, 50) mm, rotated rx 180 ry 0 rz 90 deg; joints [6.129, -45.818, 77.224, 191.643, 31.938, -189.919]
  MoveL 656 to (-890, 50, -0.5) mm, rotated rx -180 ry 0 rz 90 deg; joints [6.129, -44.378, 77.52, 191.111, 33.641, -189.286]
  MoveL 657 to (-890, 50, 50) mm, rotated rx 180 ry 0 rz 90 deg; joints [6.129, -45.818, 77.224, 191.643, 31.938, -189.919]
  MoveL 658 to (-890, 100, 50) mm, rotated rx 180 ry 0 rz 90 deg; joints [6.274, -47.892, 80.94, 191.398, 33.571, -189.535]
  MoveL 659 to (-890, 100, -0.5) mm, rotated rx 180 ry 0 rz 90 deg; joints [6.274, -46.406, 81.234, 190.897, 35.318, -188.927]
  MoveL 660 to (-890, 100, 50) mm, rotated rx 180 ry 0 rz 90 deg; joints [6.274, -47.892, 80.94, 191.398, 33.571, -189.535]
  MoveL 661 to (-890, 150, 50) mm, rotated rx -180 ry 0 rz 90 deg; joints [6.426, -49.91, 84.523, 191.216, 35.131, -189.211]
  MoveL 662 to (-890, 150, -0.5) mm, rotated rx 180 ry 0 rz 90 deg; joints [6.426, -48.376, 84.815, 190.738, 36.924, -188.62]
  MoveL 663 to (-890, 150, 50) mm, rotated rx -180 ry 0 rz 90 deg; joints [6.426, -49.91, 84.523, 191.216, 35.131, -189.211]
  MoveL 664 to (-890, 200, 50) mm, rotated rx 180 ry 0 rz 90 deg; joints [6.586, -51.879, 87.988, 191.085, 36.624, -188.936]
  MoveL 665 to (-890, 200, -0.5) mm, rotated rx -180 ry 0 rz 90 deg; joints [6.586, -50.295, 88.28, 190.626, 38.466, -188.357]
  MoveL 666 to (-890, 200, 50) mm, rotated rx 180 ry 0 rz 90 deg; joints [6.586, -51.879, 87.988, 191.085, 36.624, -188.936]
  MoveL 667 to (-890, 250, 50) mm, rotated rx 180 ry 0 rz 90 deg; joints [6.754, -53.809, 91.35, 190.999, 38.056, -188.701]
  MoveL 668 to (-890, 250, -0.5) mm, rotated rx -180 ry 0 rz 90 deg; joints [6.754, -52.173, 91.642, 190.554, 39.95, -188.129]
  MoveL 669 to (-890, 250, 50) mm, rotated rx 180 ry 0 rz 90 deg; joints [6.754, -53.809, 91.35, 190.999, 38.056, -188.701]
  MoveL 670 to (-890, 300, 50) mm, rotated rx -180 ry 0 rz 90 deg; joints [6.931, -55.705, 94.619, 190.953, 39.429, -188.502]
  MoveL 671 to (-890, 300, -0.5) mm, rotated rx -180 ry 0 rz 90 deg; joints [6.931, -54.015, 94.912, 190.519, 41.379, -187.932]
  MoveL 672 to (-890, 300, 50) mm, rotated rx -180 ry 0 rz 90 deg; joints [6.931, -55.705, 94.619, 190.953, 39.429, -188.502]
  MoveL 673 to (-890, 350, 50) mm, rotated rx -180 ry 0 rz 90 deg; joints [7.117, -57.575, 97.804, 190.942, 40.748, -188.333]
  MoveL 674 to (-890, 350, -0.5) mm, rotated rx 180 ry 0 rz 90 deg; joints [7.117, -55.827, 98.1, 190.516, 42.757, -187.761]
  MoveL 675 to (-890, 350, 50) mm, rotated rx -180 ry 0 rz 90 deg; joints [7.117, -57.575, 97.804, 190.942, 40.748, -188.333]
  MoveL 676 to (-890, 400, 50) mm, rotated rx -180 ry 0 rz 90 deg; joints [7.314, -59.424, 100.914, 190.964, 42.015, -188.191]
  MoveL 677 to (-890, 400, -0.5) mm, rotated rx -180 ry 0 rz 90 deg; joints [7.314, -57.614, 101.214, 190.543, 44.087, -187.614]
  MoveL 678 to (-890, 400, 50) mm, rotated rx -180 ry 0 rz 90 deg; joints [7.314, -59.424, 100.914, 190.964, 42.015, -188.191]
  MoveL 679 to (-890, 450, 50) mm, rotated rx -180 ry 0 rz 90 deg; joints [7.521, -61.257, 103.956, 191.017, 43.23, -188.074]
  MoveL 680 to (-890, 450, -0.5) mm, rotated rx 180 ry 0 rz 90 deg; joints [7.521, -59.382, 104.26, 190.599, 45.371, -187.489]
  MoveL 681 to (-890, 450, 50) mm, rotated rx -180 ry 0 rz 90 deg; joints [7.521, -61.257, 103.956, 191.017, 43.23, -188.074]
  MoveL 682 to (-890, 500, 50) mm, rotated rx -180 ry 0 rz 90 deg; joints [7.741, -63.08, 106.935, 191.1, 44.397, -187.98]
  MoveL 683 to (-890, 500, -0.5) mm, rotated rx -180 ry 0 rz 90 deg; joints [7.741, -61.135, 107.244, 190.682, 46.609, -187.383]
  MoveL 684 to (-890, 500, 50) mm, rotated rx -180 ry 0 rz 90 deg; joints [7.741, -63.08, 106.935, 191.1, 44.397, -187.98]
  MoveL 685 to (-890, 550, 50) mm, rotated rx -180 ry 0 rz 90 deg; joints [7.974, -64.896, 109.857, 191.212, 45.514, -187.908]
  MoveL 686 to (-890, 550, -0.5) mm, rotated rx 180 ry 0 rz 90 deg; joints [7.974, -62.877, 110.172, 190.792, 47.804, -187.296]
  MoveL 687 to (-890, 550, 50) mm, rotated rx -180 ry 0 rz 90 deg; joints [7.974, -64.896, 109.857, 191.212, 45.514, -187.908]
  MoveL 688 to (-890, 600, 50) mm, rotated rx 180 ry 0 rz 90 deg; joints [8.221, -66.711, 112.727, 191.353, 46.581, -187.858]
  MoveL 689 to (-890, 600, -0.5) mm, rotated rx -180 ry 0 rz 90 deg; joints [8.221, -64.613, 113.048, 190.929, 48.955, -187.226]
  MoveL 690 to (-890, 600, 50) mm, rotated rx 180 ry 0 rz 90 deg; joints [8.221, -66.711, 112.727, 191.353, 46.581, -187.858]
  MoveL 691 to (-890, 650, 50) mm, rotated rx -180 ry 0 rz 90 deg; joints [8.484, -68.531, 115.547, 191.524, 47.598, -187.829]
  MoveL 692 to (-890, 650, -0.5) mm, rotated rx 180 ry 0 rz 90 deg; joints [8.484, -66.347, 115.876, 191.093, 50.062, -187.174]
  MoveL 693 to (-890, 650, 50) mm, rotated rx -180 ry 0 rz 90 deg; joints [8.484, -68.531, 115.547, 191.524, 47.598, -187.829]
  MoveL 694 to (-890, 700, 50) mm, rotated rx 180 ry 0 rz 90 deg; joints [8.763, -70.36, 118.322, 191.726, 48.562, -187.821]
  MoveL 695 to (-890, 700, -0.5) mm, rotated rx -180 ry 0 rz 90 deg; joints [8.763, -68.084, 118.66, 191.286, 51.124, -187.139]
  MoveL 696 to (-890, 700, 50) mm, rotated rx 180 ry 0 rz 90 deg; joints [8.763, -70.36, 118.322, 191.726, 48.562, -187.821]
  MoveL 697 to (-890, 750, 50) mm, rotated rx 180 ry 0 rz 90 deg; joints [9.062, -72.204, 121.055, 191.96, 49.473, -187.837]
  MoveL 698 to (-890, 750, -0.5) mm, rotated rx 180 ry 0 rz 90 deg; joints [9.062, -69.829, 121.403, 191.508, 52.139, -187.123]
  MoveL 699 to (-890, 750, 50) mm, rotated rx 180 ry 0 rz 90 deg; joints [9.062, -72.204, 121.055, 191.96, 49.473, -187.837]
  MoveL 700 to (-890, 800, 50) mm, rotated rx 180 ry 0 rz 90 deg; joints [9.382, -74.07, 123.748, 192.228, 50.326, -187.877]
  MoveL 701 to (-890, 800, -0.5) mm, rotated rx -180 ry 0 rz 90 deg; joints [9.382, -71.588, 124.108, 191.762, 53.106, -187.125]
  MoveL 702 to (-890, 800, 50) mm, rotated rx 180 ry 0 rz 90 deg; joints [9.382, -74.07, 123.748, 192.228, 50.326, -187.877]
  MoveL 703 to (-890, 850, 50) mm, rotated rx -180 ry 0 rz 90 deg; joints [9.725, -75.964, 126.404, 192.533, 51.117, -187.944]
  MoveL 704 to (-890, 850, -0.5) mm, rotated rx 180 ry 0 rz 90 deg; joints [9.725, -73.365, 126.777, 192.049, 54.021, -187.147]
  MoveL 705 to (-890, 850, 50) mm, rotated rx -180 ry 0 rz 90 deg; joints [9.725, -75.964, 126.404, 192.533, 51.117, -187.944]
  MoveL 706 to (-890, 900, 50) mm, rotated rx 180 ry 0 rz 90 deg; joints [10.094, -77.894, 129.025, 192.879, 51.842, -188.041]
  MoveL 707 to (-890, 900, -0.5) mm, rotated rx -180 ry 0 rz 90 deg; joints [10.094, -75.167, 129.412, 192.373, 54.881, -187.193]
  MoveL 708 to (-890, 900, 50) mm, rotated rx 180 ry 0 rz 90 deg; joints [10.094, -77.894, 129.025, 192.879, 51.842, -188.041]
  MoveL 709 to (-890, 950, 50) mm, rotated rx -180 ry 0 rz 90 deg; joints [10.491, -79.869, 131.612, 193.27, 52.494, -188.171]
  MoveL 710 to (-890, 950, -0.5) mm, rotated rx 180 ry 0 rz 90 deg; joints [10.491, -77.003, 132.016, 192.737, 55.68, -187.263]
  MoveL 711 to (-890, 950, 50) mm, rotated rx -180 ry 0 rz 90 deg; joints [10.491, -79.869, 131.612, 193.27, 52.494, -188.171]
  MoveL 712 to (-890, 1000, 50) mm, rotated rx 180 ry 0 rz 90 deg; joints [10.921, -81.901, 134.167, 193.711, 53.065, -188.341]
  MoveL 713 to (-890, 1000, -0.5) mm, rotated rx -180 ry 0 rz 90 deg; joints [10.921, -78.881, 134.589, 193.146, 56.413, -187.362]
  MoveL 714 to (-890, 1000, 50) mm, rotated rx 180 ry 0 rz 90 deg; joints [10.921, -81.901, 134.167, 193.711, 53.065, -188.341]
  MoveL 715 to (-890, 1050, 50) mm, rotated rx -180 ry 0 rz 90 deg; joints [11.387, -84, 136.691, 194.209, 53.545, -188.556]
  MoveL 716 to (-890, 1050, -0.5) mm, rotated rx 180 ry 0 rz 90 deg; joints [11.387, -80.812, 137.134, 193.605, 57.071, -187.495]
  MoveL 717 to (-890, 1050, 50) mm, rotated rx -180 ry 0 rz 90 deg; joints [11.387, -84, 136.691, 194.209, 53.545, -188.556]
  MoveL 718 to (-890, 1100, 50) mm, rotated rx -180 ry 0 rz 90 deg; joints [11.894, -86.184, 139.185, 194.774, 53.922, -188.828]
  MoveL 719 to (-890, 1100, -0.5) mm, rotated rx 180 ry 0 rz 90 deg; joints [11.894, -82.807, 139.652, 194.122, 57.644, -187.668]
  MoveL 720 to (-890, 1100, 50) mm, rotated rx -180 ry 0 rz 90 deg; joints [11.894, -86.184, 139.185, 194.774, 53.922, -188.828]
  MoveL 721 to (-890, 1150, 50) mm, rotated rx 180 ry 0 rz 90 deg; joints [12.447, -88.469, 141.648, 195.415, 54.181, -189.167]
  MoveL 722 to (-890, 1150, -0.5) mm, rotated rx -180 ry 0 rz 90 deg; joints [12.447, -84.884, 142.143, 194.704, 58.12, -187.891]
  MoveL 723 to (-890, 1150, 50) mm, rotated rx 180 ry 0 rz 90 deg; joints [12.447, -88.469, 141.648, 195.415, 54.181, -189.167]
  MoveL 724 to (-890, 1200, 50) mm, rotated rx -180 ry 0 rz 90 deg; joints [13.054, -90.879, 144.081, 196.148, 54.302, -189.59]
  MoveL 725 to (-890, 1200, -0.5) mm, rotated rx 180 ry 0 rz 90 deg; joints [13.054, -87.061, 144.607, 195.364, 58.483, -188.174]
  MoveL 726 to (-890, 1200, 50) mm, rotated rx -180 ry 0 rz 90 deg; joints [13.054, -90.879, 144.081, 196.148, 54.302, -189.59]
  MoveL 727 to (-890, 1250, 50) mm, rotated rx 180 ry 0 rz 90 deg; joints [13.721, -93.443, 146.484, 196.991, 54.261, -190.119]
  MoveL 728 to (-890, 1250, -0.5) mm, rotated rx 180 ry 0 rz 90 deg; joints [13.721, -89.364, 147.045, 196.115, 58.71, -188.534]
  MoveL 729 to (-890, 1250, 50) mm, rotated rx 180 ry 0 rz 90 deg; joints [13.721, -93.443, 146.484, 196.991, 54.261, -190.119]
  MoveL 730 to (-890, 1300, 50) mm, rotated rx -180 ry 0 rz 90 deg; joints [14.459, -96.198, 148.853, 197.97, 54.028, -190.786]
  MoveL 731 to (-890, 1300, -0.5) mm, rotated rx -180 ry 0 rz 90 deg; joints [14.459, -91.824, 149.457, 196.976, 58.776, -188.992]
  MoveL 732 to (-890, 1300, 50) mm, rotated rx -180 ry 0 rz 90 deg; joints [14.459, -96.198, 148.853, 197.97, 54.028, -190.786]
  MoveL 733 to (-890, 1350, 50) mm, rotated rx -180 ry 0 rz 90 deg; joints [15.278, -99.19, 151.188, 199.119, 53.564, -191.634]
  MoveL 734 to (-890, 1350, -0.5) mm, rotated rx 180 ry 0 rz 90 deg; joints [15.278, -94.484, 151.841, 197.973, 58.646, -189.581]
  MoveL 735 to (-890, 1350, 50) mm, rotated rx -180 ry 0 rz 90 deg; joints [15.278, -99.19, 151.188, 199.119, 53.564, -191.634]
  MoveL 736 to (-890, 1400, 50) mm, rotated rx -180 ry 0 rz 90 deg; joints [16.194, -102.482, 153.485, 200.489, 52.821, -192.724]
  MoveL 737 to (-890, 1400, -0.5) mm, rotated rx 180 ry 0 rz 90 deg; joints [16.194, -97.401, 154.196, 199.141, 58.271, -190.344]
  MoveL 738 to (-890, 1400, 50) mm, rotated rx -180 ry 0 rz 90 deg; joints [16.194, -102.482, 153.485, 200.489, 52.821, -192.724]
  MoveL 739 to (-890, 1450, 50) mm, rotated rx -180 ry 0 rz 110 deg; joints [23.693, -102.084, 153.222, 230.82, 63.02, -209.102]
  MoveL 740 to (-890, 1450, -0.5) mm, rotated rx -180 ry 0 rz 110 deg; joints [23.693, -97.049, 153.926, 228.762, 66.728, -204.262]
  MoveL 741 to (-890, 1450, 50) mm, rotated rx -180 ry 0 rz 110 deg; joints [23.693, -102.084, 153.222, 230.82, 63.02, -209.102]
  MoveL 742 to (-960, 50, 50) mm, rotated rx 180 ry 0 rz 90 deg; joints [7.973, -45.453, 76.566, 195.165, 32.019, -192.942]
  MoveL 743 to (-960, 50, -0.5) mm, rotated rx -180 ry 0 rz 90 deg; joints [7.973, -44.021, 76.864, 194.48, 33.691, -192.127]
  MoveL 744 to (-960, 50, 50) mm, rotated rx 180 ry 0 rz 90 deg; joints [7.973, -45.453, 76.566, 195.165, 32.019, -192.942]
  MoveL 745 to (-960, 100, 50) mm, rotated rx -180 ry 0 rz 90 deg; joints [8.161, -47.53, 80.293, 194.842, 33.654, -192.439]
  MoveL 746 to (-960, 100, -0.5) mm, rotated rx 180 ry 0 rz 90 deg; joints [8.161, -46.052, 80.587, 194.196, 35.369, -191.655]
  MoveL 747 to (-960, 100, 50) mm, rotated rx -180 ry 0 rz 90 deg; joints [8.161, -47.53, 80.293, 194.842, 33.654, -192.439]
  MoveL 748 to (-960, 150, 50) mm, rotated rx -180 ry 0 rz 90 deg; joints [8.358, -49.548, 83.882, 194.6, 35.216, -192.014]
  MoveL 749 to (-960, 150, -0.5) mm, rotated rx 180 ry 0 rz 90 deg; joints [8.358, -48.023, 84.175, 193.984, 36.977, -191.252]
  MoveL 750 to (-960, 150, 50) mm, rotated rx -180 ry 0 rz 90 deg; joints [8.358, -49.548, 83.882, 194.6, 35.216, -192.014]
  MoveL 751 to (-960, 200, 50) mm, rotated rx 180 ry 0 rz 90 deg; joints [8.565, -51.516, 87.353, 194.426, 36.712, -191.652]
  MoveL 752 to (-960, 200, -0.5) mm, rotated rx -180 ry 0 rz 90 deg; joints [8.565, -49.942, 87.644, 193.834, 38.521, -190.906]
  MoveL 753 to (-960, 200, 50) mm, rotated rx 180 ry 0 rz 90 deg; joints [8.565, -51.516, 87.353, 194.426, 36.712, -191.652]
  MoveL 754 to (-960, 250, 50) mm, rotated rx 180 ry 0 rz 90 deg; joints [8.782, -53.444, 90.717, 194.31, 38.147, -191.343]
  MoveL 755 to (-960, 250, -0.5) mm, rotated rx -180 ry 0 rz 90 deg; joints [8.782, -51.818, 91.009, 193.738, 40.007, -190.606]
  MoveL 756 to (-960, 250, 50) mm, rotated rx 180 ry 0 rz 90 deg; joints [8.782, -53.444, 90.717, 194.31, 38.147, -191.343]
  MoveL 757 to (-960, 300, 50) mm, rotated rx 180 ry 0 rz 90 deg; joints [9.01, -55.337, 93.986, 194.245, 39.525, -191.08]
  MoveL 758 to (-960, 300, -0.5) mm, rotated rx 180 ry 0 rz 90 deg; joints [9.01, -53.657, 94.279, 193.687, 41.44, -190.347]
  MoveL 759 to (-960, 300, 50) mm, rotated rx 180 ry 0 rz 90 deg; joints [9.01, -55.337, 93.986, 194.245, 39.525, -191.08]
  MoveL 760 to (-960, 350, 50) mm, rotated rx -180 ry 0 rz 90 deg; joints [9.25, -57.202, 97.171, 194.227, 40.85, -190.857]
  MoveL 761 to (-960, 350, -0.5) mm, rotated rx 180 ry 0 rz 90 deg; joints [9.25, -55.465, 97.466, 193.679, 42.822, -190.122]
  MoveL 762 to (-960, 350, 50) mm, rotated rx -180 ry 0 rz 90 deg; joints [9.25, -57.202, 97.171, 194.227, 40.85, -190.857]
  MoveL 763 to (-960, 400, 50) mm, rotated rx 180 ry 0 rz 90 deg; joints [9.504, -59.044, 100.278, 194.251, 42.123, -190.668]
  MoveL 764 to (-960, 400, -0.5) mm, rotated rx 180 ry 0 rz 90 deg; joints [9.504, -57.247, 100.577, 193.711, 44.157, -189.928]
  MoveL 765 to (-960, 400, 50) mm, rotated rx 180 ry 0 rz 90 deg; joints [9.504, -59.044, 100.278, 194.251, 42.123, -190.668]
